// TwinCAT 3 PLC project Area2
// ProgramVersion: 3.1.4023.0
// libraries:
//   Tc2_DataExchange, * (Beckhoff Automation GmbH)
//   Tc2_EtherCAT, * (Beckhoff Automation GmbH)
//   Tc2_MC2, * (Beckhoff Automation GmbH)
//   Tc2_Standard, * (Beckhoff Automation GmbH)
//   Tc2_System, * (Beckhoff Automation GmbH)
//   Tc2_TcpIp, * (Beckhoff Automation GmbH)
//   Tc2_Utilities, * (Beckhoff Automation GmbH)
//   Tc3_BA_Common, * (Beckhoff Automation GmbH)
//   Tc3_Database, * (Beckhoff Automation GmbH)
//   Tc3_JsonXml, * (Beckhoff Automation GmbH)
//   Tc3_Module, * (Beckhoff Automation GmbH)
//   Tc3_PackML_V2, * (Beckhoff Automation GmbH)
// project tree:
//   COMs/Comms_ADS/ AdsData.TcDUT, AdsMessage.TcDUT, AdsMessageQueue.TcPOU, AdsSocket.TcPOU, AdsTcpUnitEx.TcPOU
//   COMs/Comms_TCP/ TcpServer1Vision.TcPOU (not stored), VisionFrame.TcDUT, VisionSuite.TcDUT
//   COMs/Comms_TCP/Types/ TcpData.TcDUT (not stored), TcpDataQueue.TcPOU (not stored)
//   COMs/Local Devices/ EcNetwork.TcPOU
//   COMs/ Watchdog.TcPOU
//   DUTs/Enums/ AreaEnum.TcDUT, E_PMLCustomUnitMode.TcDUT (not stored), SectionEnum.TcDUT, SectionTask.TcDUT, Cover.TcDUT (not stored), EventsEnum.TcTLEO, MaterialEnum.TcDUT, MaterialType.TcDUT (not stored), Surface.TcDUT (not stored)
//   DUTs/Enums/Materials/ Cardboard.TcDUT (not stored), Chipboard.TcDUT (not stored), CornerGuard.TcDUT (not stored), WoodBunk.TcDUT
//   DUTs/Hardware/ A21ToolStorage.TcDUT, FoldingMachine.TcDUT (not stored), PMLStackLight.TcPOU, ToolStorage.TcDUT
//   DUTs/Hardware/Big Machines/ StrapMachine.TcPOU, WrapMachine.TcPOU (not stored)
//   DUTs/Hardware/Conveyors/ Conveyor.TcPOU, ConveyorLSC.TcPOU (not stored), ConveyorMode.TcDUT (not stored), ConveyorSC.TcPOU, ConveyorSC_NC.TcPOU
//   DUTs/Hardware/Insertion Package/Drives/ AirPiston.TcPOU, ClearLinkMC.TcPOU (not stored), ServoNC.TcPOU, SimplePiston.TcPOU (not stored)
//   DUTs/Hardware/Insertion Package/ Homing.TcDUT (not stored), Insertion.TcPOU, SuctionPad.TcDUT
//   DUTs/Hardware/Insertion Package/Prototypes/ FBA_Drive.TcPOU (not stored), FBA_TrifectaDrive.TcPOU, I_ContinuousDrive.TcIO (not stored), I_Drive.TcIO, I_EncodedDrive.TcIO (not stored), I_PositionalDrive.TcIO
//   DUTs/Hardware/Material Holders/ MaterialHolder.TcPOU (not stored), MaterialSlot.TcDUT (not stored), SkidMagazine.TcPOU, StagingTable.TcPOU (not stored)
//   DUTs/Hardware/Robots/ I_Area2Robot.TcIO, KukaRobot.TcPOU, RobotA21.TcPOU, RobotA26.TcPOU, RobotA22.TcPOU
//   DUTs/Hardware/Robots/Tasks/ TaskA21.TcDUT (not stored), TaskA22.TcDUT (not stored), TaskA26.TcDUT
//   DUTs/Bundle/ Bundle.TcDUT, CardboardMaterial.TcDUT (not stored), Interval.TcDUT (not stored), Material.TcDUT (not stored), PositionMaterials.TcDUT
//   DUTs/Containers/ DynamicQueue.TcPOU (not stored), PtrQueue.TcPOU, IntQueue.TcPOU (not stored), Queue.TcPOU (not stored), StringQueue.TcPOU (not stored)
//   EventLogging/ EventLogger.TcIO (not stored), SqlDatabaseAccessor.TcPOU
//   / GlobalTextList.TcGTLO (not stored), PlcTask.TcTTO
//   GVLs/ COM.TcGVL, GVL.TcGVL, CONSTS.TcGVL
//   HARDWARE_DISTRUBUTION/ A24_A26.TcPOU, ConveyorSyncUnit.TcPOU, GenericSubarea.TcPOU, A21.TcPOU, A22.TcPOU, A23.TcPOU (not stored), A24.TcPOU, A25.TcPOU, A26.TcPOU (not stored)
//   POUs/Helper Functions/Document/ CreateJsonDocumentManual.TcPOU (not stored), CreateJsonDocumentAuto.TcPOU, FrameIsValid.TcPOU, VisionJsonParser.TcPOU (not stored)
//   POUs/Helper Functions/General/ BufferIsEmpty.TcPOU (not stored), BundleIsValid.TcPOU (not stored), InRange.TcPOU, PositionIsValid.TcPOU (not stored), TimestructToString.TcPOU (not stored), WithinTolerance.TcPOU
//   POUs/Helper Functions/Hardware Modules/ CheckEcNetwork.TcPOU, InsertionQuality.TcPOU, SetSuctions.TcPOU (not stored), SetSuctionsPtr.TcPOU (not stored), SetupHardware.TcPOU (not stored), SuctionQuality.TcPOU, SuctionQualityPtr.TcPOU (not stored)
//   POUs/Helper Functions/Material Functions/ GetPairMasterLength.TcPOU (not stored), GetMaterialLength.TcPOU, MatchesMaterialType.TcPOU
//   POUs/Helper Functions/Data Manipulation/ AddToStringArray.TcPOU, ArrayContains.TcPOU, DataIsEmpty.TcPOU (not stored), CleanStringsArray.TcPOU (not stored), IntegerBitAccess.TcPOU (not stored), IntegerToBoolArray.TcPOU (not stored), JoinStrings.TcPOU
//   POUs/ MAIN.TcPOU, TypeSizeCheck.TcPOU
//   Sections/A21a - Chipboard/AOIs/ AOI_LoadChipboard.TcPOU (not stored)
//   Sections/A21a - Chipboard/ ChipboardEx.TcPOU
//   Sections/A21b - Wood Bunk/AOIs/ AOI_LoadWoodBunk.TcPOU (not stored), AOI_StageWoodBunk.TcPOU, AOI_StagingTemplate.TcPOU (not stored)
//   Sections/A21b - Wood Bunk/ WoodBunkEx.TcPOU
//   Sections/A22 - Cardboard/AOIs/ AOI_LoadCornerCardboard.TcPOU (not stored), AOI_LoadCornerGuard.TcPOU (not stored), AOI_LoadFlatCardboard.TcPOU (not stored)
//   Sections/A22 - Cardboard/ CardboardEx.TcPOU
//   Sections/A26 - Spacer Recollection/ SpacerRecollectionUnit.TcPOU
//   Sections/Abstract/ SectionEx.TcPOU
// real-time tasks:
//   TASK PlcTask: cycle T#10ms, priority 20, ADS port 350
// motion (NC):
//   TASK NC-Task 1 SAF: cycle T#2ms, priority 4, ADS port 501
//   TASK NC-Task 1 SVB: cycle T#10ms, priority 8, ADS port 511
//   AXIS Axis 1 (id 1)
//     OtherSettings: AllowMotionCmdToSlave=true
//     encoder EncType=19
//       EncPara: MaxCount=#xffffffff
//     drive DrvType=16
//       DrvPara: MaxCount=#xffffffff, DriveControlDWord=#x00000100
//         Analog: TorqueSetpointScale=10, ScaleFactorActTorque=0.1
//         TimeComp: TaskDelayCycles=1
//     controller CtrType=1
//       CtrPara: PriorControlFactor=1
//         Observer: BandWidth=20
// I/O:
//   DEVICE Device 1 (EtherCAT) (disabled), AmsNetId 192.168.101.188.2.1
//     Term 1 (EK1200) [EK1200-5000 EtherCAT Power supply (2A E-Bus)]
//       Term 2 (EL2809) [EL2809 16Ch. Dig. Output 24V, 0.5A]
//       Term 3 (EL9011) [EL9011 End Terminal]
//   DEVICE Device 4 (EtherCAT) (disabled), AmsNetId 192.168.101.188.5.1
//     Drive 4 (CDHD) [CDHD EtherCAT Drive (CoE)]
// variable links:
//   NC-Task 1 SAF/Axes/Axis 1 <-> Device 4 (EtherCAT)/Drive 4 (CDHD)
//     Drive/Inputs/In/nDataIn1 <-> TxPDO 4/Following Error Actual Value
//     Drive/Inputs/In/nDataIn3[0] <-> TxPDO 1/Torque Actual Value
//     Drive/Inputs/In/nDcOutputTime <-> InfoData/DcOutputShift
//     Drive/Inputs/In/nState1 <-> TxPDO 1/StatusWord
//     Drive/Inputs/In/nState2 <-> TxPDO 1/StatusWord @bit 8
//     Drive/Inputs/In/nState4 @bit 1 <-> WcState/InputToggle
//     Drive/Inputs/In/nState4 <-> WcState/WcState
//     Drive/Inputs/In/nState5 <-> TxPDO 1/Modes of operation display
//     Drive/Outputs/Out/nCtrl1 <-> RxPDO 1/ControlWord
//     Drive/Outputs/Out/nCtrl2 <-> RxPDO 1/ControlWord @bit 8
//     Drive/Outputs/Out/nCtrl5 <-> RxPDO 1/Modes of operation
//     Drive/Outputs/Out/nDataOut1 <-> RxPDO 2/Target position
//     Drive/Outputs/Out/nDataOut2 <-> RxPDO 3/Target Velocity
//     Drive/Outputs/Out/nDataOut3[0] <-> RxPDO 4/Torque Offset
//     Drive/Outputs/Out/nDataOut4[0] <-> RxPDO 4/Target torque
//     Enc/Inputs/In/nDataIn1 <-> TxPDO 2/Position actual value
//     Enc/Inputs/In/nDcInputTime <-> InfoData/DcInputShift
//     Enc/Inputs/In/nState4 @bit 1 <-> WcState/InputToggle
//     Enc/Inputs/In/nState4 <-> WcState/WcState

CONFIGURATION Area2
    RESOURCE PLC ON TwinCAT3
        TASK PlcTask(INTERVAL := T#10ms, PRIORITY := 20);
        PROGRAM MAIN WITH PlcTask : MAIN;
    END_RESOURCE
END_CONFIGURATION

// ---- COMs/Comms_ADS/AdsData.TcDUT
{attribute 'enable_dynamic_creation'}
TYPE AdsData :
STRUCT
	description : EventsEnum; //purpose
	
	timestamp : TIMESTRUCT; //relevant timestamp (ex: arrival time)
	
	binaryData : ARRAY[0..100000] OF BYTE; //contents
END_STRUCT
END_TYPE

// ---- COMs/Comms_ADS/AdsMessage.TcDUT
{attribute 'enable_dynamic_creation'}
TYPE AdsMessage :
STRUCT
	recipient : STRING;
	contents : AdsData;
END_STRUCT
END_TYPE

// ---- COMs/Comms_TCP/VisionFrame.TcDUT
TYPE VisionFrame :
STRUCT
	MaterialID : STRING;
	CheckFor : STRING;
	CameraNumber : DINT;
	
	SuccessFlag : DINT;
	OrientAdjustX : LREAL;
	OrientAdjustY : LREAL;
	OrientAdjustZ : LREAL;
END_STRUCT
END_TYPE

// ---- COMs/Comms_TCP/VisionSuite.TcDUT
TYPE VisionSuite :
STRUCT
	json : STRING(1000);
	frame : VisionFrame;
	data : TcpData;
END_STRUCT
END_TYPE

// ---- DUTs/Enums/AreaEnum.TcDUT
{attribute 'qualified_only'}
{attribute 'to_string'}
TYPE AreaEnum :
(
	NULL_AREA,
	
	AREA_1,
	AREA_2,
	AREA_3,
	AREA_4,
	AREA_5,
	AREA_6,
	
	size
	
);
END_TYPE
(*
when generating AdsMessage types, use TO_STRING to convert these enums to a recipient string
*)

// ---- DUTs/Enums/Materials/WoodBunk.TcDUT
{attribute 'qualified_only'}
{attribute 'to_string'}
TYPE WoodBunk : //21
(
	WDW20 := 1, //special top (wide) 
	WDW22,

	WDT20, //top
	WDT22, 
	WDT28,

	WDB20, //bottom
	WDB22, 
	WDB28, 

	WDS08, //side
	WDS10, 
	WDS12, 
	WDS14, 
	WDS20, 
	WDS22, 
	WDS28, 
	
	size
	(*
	WDS08_WDS08, //side combined - X - 2 wood bunks joined by underscore
	WDS08_WDS10, 
	WDS12_WDS12, 
	WDS12_WDS14, 
	WDS20_WDS10, 
	WDS20_WDS12, 
	
	sizeAll
	*)
);
END_TYPE

// ---- DUTs/Enums/SectionEnum.TcDUT
{attribute 'qualified_only'}
{attribute 'to_string'}
TYPE SectionEnum :
(
	NULL_SECTION,
	
	PAPER,
	CARDBOARD_CORNERGUARD,
	CHIPBOARD,
	WOOD_BUNK,
	OUTPUT,
	
	SPACER_RECOLLECTOR,
	
	size
);
END_TYPE

// ---- DUTs/Hardware/A21ToolStorage.TcDUT
TYPE A21ToolStorage :
STRUCT
	pos1ChipboardEOAT AT %I* : BOOL;
	pos1WoodBunkEOAT AT %I* : BOOL;
	
	pos2ChipboardEOAT AT %I* : BOOL;
	pos2WoodBunkEOAT AT %I* : BOOL;
END_STRUCT
END_TYPE

// ---- DUTs/Hardware/Insertion Package/SuctionPad.TcDUT
TYPE SuctionPad :
STRUCT
	enable AT %Q* : BOOL;
	occupied AT %I* : BOOL;
END_STRUCT
END_TYPE

// ---- DUTs/Hardware/Robots/Tasks/TaskA26.TcDUT
{attribute 'qualified_only'}
{attribute 'to_string'}
//{attribute 'strict'}
TYPE TaskA26 :
(
	IDLE,
	PICK_SPACER,
	MEASURE,
	
	size
);
END_TYPE

// ---- DUTs/Hardware/ToolStorage.TcDUT
TYPE ToolStorage :
STRUCT
	eoatA_pos1 : BOOL;
	eoatB_pos1 : BOOL;
	
	eoatA_pos2 : BOOL;
	eoatB_pos2 : BOOL;	
END_STRUCT
END_TYPE

// ---- DUTs/Bundle/Bundle.TcDUT
{attribute 'enable_dynamic_creation'}
TYPE Bundle :
STRUCT
	id : STRING;
	weight : REAL;
	
	length : INT;
	width : INT;
	height : INT;
	
	pieces : INT;
	layers : INT;
	piecesPerLayer : INT;
	
	extrusionWeight : INT;
	extrusionHeight : INT;
	extrusionWidth : INT;
	
	//if a process is true, send it to the correct area and turn it false when complete
	reqProcesses : ARRAY[0..3] OF BOOL;
	
	manRE, autoRE : BOOL; //repacking - coming soon
	manSS, autoSS : BOOL; //packaging
	
	currStep : USINT; //for runtime use only
	
	paperFront : BOOL;
	paperBack : BOOL;
	cardboardFront : BOOL;
	cardboardBack : BOOL;
	
	paperTop : ARRAY[0..CONSTS.maxPairs] OF Interval;
	paperLeft : ARRAY[0..CONSTS.maxPairs] OF Interval;
	paperRight : ARRAY[0..CONSTS.maxPairs] OF Interval;
	paperBottom : ARRAY[0..CONSTS.maxPairs] OF Interval;
		
	cardboard : ARRAY[0..CONSTS.maxPairs] OF PositionMaterials;
	cardboardFolds : ARRAY[Surface.TOP_LEFT..Surface.BOTTOM_RIGHT] OF ARRAY[0..CONSTS.maxPairs] OF INT;
	
	topLeftFolds : ARRAY[0..CONSTS.maxPairs] OF INT;
	topRightFolds : ARRAY[0..CONSTS.maxPairs] OF INT;
	bottomLeftFolds : ARRAY[0..CONSTS.maxPairs] OF INT;
	bottomRightFolds : ARRAY[0..CONSTS.maxPairs] OF INT;
	
	cornerGuard : ARRAY[0..CONSTS.maxPairs] OF PositionMaterials;
	
	chipboard : ARRAY[0..CONSTS.maxPairs] OF PositionMaterials;
	woodBunk : ARRAY[0..CONSTS.maxPairs] OF PositionMaterials;
	
	cardboard_over_cornerGuard : BOOL;
	
	//for production log database
	bypass : BOOL;
	
	timeStart : TIMESTRUCT;
	timeDone : TIMESTRUCT;
END_STRUCT
END_TYPE

// ---- DUTs/Bundle/PositionMaterials.TcDUT
TYPE PositionMaterials : //REMOVE FOLDING INFORMATION FROM THIS STRUCTURE AND PLACE IN BUNDLE
STRUCT
	position : REAL; //:= GVL.nullPos; //default value is set to predefined constant if bundle needs less than 32 position material pairs
	
	top : STRING;
	right : STRING;
	left : STRING;
	//sides : STRING;
	bottom : STRING;
	
	topLeft : STRING;
	//topLeftFold : USINT;
	
	topRight : STRING;
	//topRightFold : USINT;
	
	bottomLeft : STRING;
	//bottomLeftFold : USINT;
	
	bottomRight : STRING;
	//bottomRightFold : USINT;

	wrapPoints : USINT;
	wrapRotations : USINT;
END_STRUCT
END_TYPE

// ---- DUTs/Enums/SectionTask.TcDUT
{attribute 'qualified_only'}
//{attribute 'strict'}
TYPE SectionTask :
(
	IDLE,
	ALIGNING,
	ACTIVE,
	DISCHARGE,
	COMPLETE,
	
	size
);
END_TYPE

// ---- DUTs/Enums/EventsEnum.TcTLEO
{attribute 'qualified_only'}
{attribute 'strict'}
{attribute 'to_string'}
TYPE EventsEnum :
(
	NO_EVENT,
	TEST_COMMS, 
	
	//standard operation
	BUNDLE_ETA,
	BUNDLE_IN,
	BUNDLE_OUT,
	BUNDLE_RECEIVED,
	BUNDLE_COMPLETE,
	
	//area complete
	AREA_1_COMPLETE,
	AREA_2_COMPLETE,
	AREA_3_COMPLETE,
	AREA_4_COMPLETE,
	AREA_5_COMPLETE,
	AREA_6_COMPLETE,
	
	//area specific operations
	SECTION_PAPER_COMPLETE,
	SECTION_CARDBOARD_CORNERGUARD_COMPLETE,
	SECTION_CHIPBOARD_COMPLETE,
	SECTION_WOODBUNK_COMPLETE,

	//standard errors
	BACKLOG,
	MACHINE_FAILURE,
	DELAY,
	BUNDLE_EARLY_RECEIVED,
	BUNDLE_LATE_RECEIVED,
	
	//area specific errors
	SECTION_PAPER_FAIL,
	SECTION_CARDBOARD_CORNERGUARD_FAIL,
	SECTION_CHIPBOARD_FAIL,
	SECTION_WOODBUNK_FAIL,
	
	//robots, motors, database, connections, etc
	
	size
);
END_TYPE

// ---- DUTs/Enums/MaterialEnum.TcDUT
{attribute 'qualified_only'}
{attribute 'strict'}
{attribute 'to_string'}
TYPE MaterialEnum :
(
	//CARDBOARD - 6 x 3
	CAR20S, CAR20M, CAR20L, CAR28S, CAR28M, CAR28L, //base (flat)
	CAR20SF, CAR20MF, CAR20LF, CAR28SF, CAR28MF, CAR28LF, //single folded (L shape) - F
	CAR20SD, CAR20MD, CAR20LD, CAR28SD, CAR28MD, CAR28LD, //double folded (C shape) - D
	
	//CHIPBOARD - 2
	CIP18, CIP54,
	
	//CORNER BOARD - 2
	COR48, COR96,
	
	//PAPER - 1
	PAP28,
	
	//WOOD BUNK - 21
	WDT20, WDT22, WDT28, //top
	WDB20, WDB22, WDB28, //bottom
	WDS08, WDS10, WDS12, WDS14, WDS20, WDS22, WDS28, //side
	WDS8X8, WDS8X10, WDS12X12, WDS12X14, WDS20X10, WDS20X12, //side combined - X
	WDW20, WDW22, //special top (wide)
	
	size //number of materials
);
END_TYPE

// ---- GVLs/COM.TcGVL
{attribute 'qualified_only'}
VAR_GLOBAL
	adsMajorNetwork : AdsTcpUnitEx;
END_VAR

// ---- GVLs/GVL.TcGVL
{attribute 'qualified_only'}
VAR_GLOBAL
	bundleOut : Bundle; //may or may not be used?
	
	iecCriticalSection : FB_IecCriticalSection; //if communication is separated into their own core/task
END_VAR
VAR_GLOBAL //changed from PROGRAMs to global instances of FUNCTION_BLOCKs to enable inheritance
	sa21 : A21;
	sa22 : A22;
	sa23 : A23;
	sa24 : A24;
	sa25 : A25;
	sa26 : A26;
END_VAR

// ---- GVLs/CONSTS.TcGVL
{attribute 'qualified_only'}
VAR_GLOBAL CONSTANT
	maxPairs : USINT := 16;
	initArraySize : USINT := 4;
	maxQueue : INT := 16;
	
	nullPos : REAL := -1;
	
	numMaterials : INT := 32;
	allMaterials : ARRAY[0..numMaterials] OF Material := [
		(code := '', width := 0, length := 0), //null material
		(code := 'PAP28', width := 28, length := -1),
		
		(code := 'CAR20S', width := 20, length := 30),
		(code := 'CAR20M', width := 20, length := 45),
		(code := 'CAR20L', width := 20, length := 60),
		(code := 'CAR28S', width := 28, length := 30),
		(code := 'CAR28M', width := 28, length := 45),
		(code := 'CAR28L', width := 28, length := 60),
		
		(code := 'COR48', width := 1.5, length := 48),
		(code := 'COR96', width := 1.5, length := 96),
		
		(code := 'CIP18', width := 20, length := 18),
		(code := 'CIP54', width := 20, length := 54),
		
		(code := 'WDT20', width := 20, length := 2.5),
		(code := 'WDT22', width := 22, length := 2.5),
		(code := 'WDT28', width := 28, length := 2.5),
		
		(code := 'WDB20', width := 20, length := 2.5),
		(code := 'WDB22', width := 22, length := 2.5),
		(code := 'WDB28', width := 28, length := 2.5),
		
		(code := 'WDS08', width := 8, length := 2.5),
		(code := 'WDS10', width := 10, length := 2.5),
		(code := 'WDS12', width := 12, length := 2.5),
		(code := 'WDS14', width := 14, length := 2.5),
		(code := 'WDS8x8', width := 16, length := 2.5),
		(code := 'WDS8x10', width := 18, length := 2.5),
		(code := 'WDS20', width := 20, length := 2.5),
		(code := 'WDS22', width := 22, length := 2.5),
		(code := 'WDS12x12', width := 24, length := 2.5),
		(code := 'WDS12x14', width := 26, length := 2.5),
		(code := 'WDS28', width := 28, length := 2.5),
		(code := 'WDS20x10', width := 30, length := 2.5),
		(code := 'WDS20x12', width := 32, length := 2.5),
		
		(code := 'WDW20', width := 20, length := 6),
		(code := 'WDW22', width := 22, length := 6)];
		
	precisionTolerance : REAL := 0.05 * 25.4;
END_VAR

// ---- DUTs/Hardware/Insertion Package/Prototypes/I_Drive.TcIO
INTERFACE I_Drive

{attribute 'monitoring':='call'}
PROPERTY Active : BOOL
GET
END_GET
END_PROPERTY

{attribute 'monitoring':='call'}
PROPERTY AtHome : BOOL
GET
END_GET
END_PROPERTY

{attribute 'monitoring':='call'}
PROPERTY Error : BOOL
GET
END_GET
END_PROPERTY

{attribute 'monitoring':='call'}
PROPERTY HomeSet : BOOL
GET
END_GET
END_PROPERTY

METHOD ABSTRACT homingSequence : BOOL
VAR_INPUT
END_VAR
END_METHOD

METHOD reset : BOOL
VAR_INPUT
END_VAR
END_METHOD

METHOD ABSTRACT stop : BOOL
VAR_INPUT
END_VAR
END_METHOD

METHOD toHome : BOOL
VAR_INPUT
END_VAR
END_METHOD

END_INTERFACE

// ---- DUTs/Hardware/Insertion Package/Prototypes/I_PositionalDrive.TcIO
INTERFACE I_PositionalDrive EXTENDS I_Drive

PROPERTY CurrentPosition : LREAL
GET
END_GET
SET
END_SET
END_PROPERTY

METHOD ABSTRACT moveAbsolute : BOOL
VAR_INPUT
	newTarget : LREAL; 
END_VAR
END_METHOD

METHOD ABSTRACT moveRelative : BOOL
VAR_INPUT
	distance : LREAL;
END_VAR
END_METHOD

PROPERTY TargetPosition : LREAL
GET
END_GET
SET
END_SET
END_PROPERTY

END_INTERFACE

// ---- DUTs/Hardware/Robots/I_Area2Robot.TcIO
INTERFACE I_Area2Robot
(*
currently all robots use 20-WORD arrays inputs and outputs so they extend from KukaRobot
if robot IOs are replaced with specific data types for each subarea, they should implement this interface instead
*)

//{attribute 'monitoring' := 'variable'}
{attribute 'monitoring' := 'call'}
PROPERTY Busy : BOOL
GET
END_GET
END_PROPERTY

METHOD clearCommand : BOOL
VAR_INPUT
END_VAR
END_METHOD

//{attribute 'monitoring' := 'variable'}
{attribute 'monitoring' := 'call'}
PROPERTY Done : BOOL
GET
END_GET
END_PROPERTY

{attribute 'monitoring' := 'call'}
PROPERTY Ready : BOOL
GET
END_GET
END_PROPERTY

METHOD release : BOOL
VAR_INPUT
	sectionReservation : SectionEnum;
END_VAR
END_METHOD

METHOD reserve : BOOL
VAR_INPUT
	reserveRequest : SectionEnum;
END_VAR
(*
this method exists because chipboard and wood bunk operations use the same robot
both sections need to check if the robot is open to commands before use
*)
END_METHOD

{attribute 'monitoring' := 'call'}
PROPERTY Reserved : BOOL
GET
END_GET
END_PROPERTY

METHOD reset : BOOL
END_METHOD

METHOD stop : BOOL
VAR_INPUT
END_VAR
END_METHOD

END_INTERFACE

// ---- POUs/MAIN.TcPOU
PROGRAM MAIN
VAR_OUTPUT //globally readable, but only modifiable by MAIN
	outputBufferPass, outputBufferFail : Bundle;
	numOutputBundles : USINT := 0;
	
	bundleIn : Bundle;
	bundleOut : Bundle;
	
	start : BOOL;
	
	ready : BOOL;
	busy : BOOL;
	done : BOOL;
	error : BOOL;
	backlog : BOOL;
	
	stop : BOOL;
	execute : BOOL;
	hold : BOOL;
	reset : BOOL;
	
	localTime : TIMESTRUCT;
	
	pmlMode : E_PMLCustomUnitMode;
	pmlState : E_PMLState;
	pmlModeString : STRING;
	pmlStateString : STRING;
END_VAR
VAR
	clearPassBuffer, clearFailBuffer AT %I* : BOOL;
	receiverStruct : AdsData;
	
	//ETA is not strictly required, area will process bundle even if it is not in ETA arrays
	expectedBundles : ARRAY[0..CONSTS.maxQueue] OF STRING; //bundles expected to arrive
	expectedArrivals : ARRAY[0..CONSTS.maxQueue] OF TIMESTRUCT; //bundles expected to arrive
	numEtaBundles : INT;
	
	//parallel arrays - bundle, bypass
	numBundles : INT;
	bundlesQueue : ARRAY[0..CONSTS.maxQueue] OF Bundle;
END_VAR
VAR //sections
	spacerRecollector : SpacerRecollectionUnit;
	//paperSection : PaperEx;
	cardboardSection : CardboardEx;
	chipboardSection : ChipboardEx;
	woodBunkSection : WoodBunkEx;
	//outputSection : AreaOutputEx;	
END_VAR
VAR
	ecDiagnostics_EK1200 : EcNetwork;
	
	fbLocalSystemTime : FB_LocalSystemTime;
	dbLogger : SqlDatabaseAccessor;
	
	pmlCommand : E_PMLCommand;
	pmlStateMachine : PML_StateMachine;
	
	pmlModeRequest : E_PMLCustomUnitMode := ePMLCustomUnitMode_Production;
	pmlModeManager : PML_UnitModeManager;
	
	processModes : (CONCURRENT, SINGLE, SERIAL);
	(*
	COCURRENT - cram as many bundles as can fit in the cell
	SINGLE - 1 bundle in the cell at a time, can be processed by many sections at the same time
	SERIAL - 1 bundle in the cell at a time, 1 section a time
		after completing a section, align bundle to action point of next section
	*)
END_VAR
VAR //these variables are only tracked for HMI
	sectionsBusy : ARRAY[0..SectionEnum.size] OF BOOL;
	sectionsIterator : ARRAY[0..SectionEnum.size] OF INT;
END_VAR
VAR
	cycleTime : DWORD;
	maxCycle : DWORD;
	masterProfiler : Profiler;
END_VAR

TypeSizeCheck();
masterProfiler(START:= TRUE, RESET:= , BUSY=> , DATA=> );

(*
Area 2 is ready when:
	no conveyors in A2.4 are occupied
	robot in A2.6 is not busy
if Area 2 is not ready, dispatch PLC must block operator from sending bundles here
*)

(*
busy := paperSection.busy OR cardboardCornerGuardSection.busy OR chipboardSection.busy OR woodBunkSection.busy OR outputSection.busy;
done := outputSection.done;
backlog := numBundlesQueue > 5;
*)

initSections();

blocks();

runPML();

runSubareas();

IF
	COM.adsMajorNetwork.fetchData(
		senderName := TO_STRING(AreaEnum.AREA_3), 
		data => receiverStruct)
THEN
	interpretTransmission(receiverStruct);
END_IF

IF ready AND BundleIsValid(bundleIn) THEN
	receive();
END_IF

IF clearPassBuffer OR clearFailBuffer THEN
	transfer();
	shiftBundles();
END_IF

dbLogger();

masterProfiler(START:= FALSE, RESET:= , BUSY=> , DATA=> );
cycleTime := masterProfiler.DATA.LastExecTime;
maxCycle := masterProfiler.DATA.MaxExecTime;

METHOD PRIVATE blocks : BOOL
fbLocalSystemTime(
	sNetID:= '', 
	bEnable:= TRUE, 
	dwCycle:= , 
	dwOpt:= , 
	tTimeout:= , 
	bValid=> , 
	systemTime=> localTime, 
	tzID=> );
	
ecDiagnostics_EK1200(
	enable:= TRUE, 
	netID:= , 
	slaves=> , 
	slaveStates=> , 
	deviceIndexesA21=> , 
	deviceIndexesA22=> , 
	deviceIndexesA23=> , 
	deviceIndexesA24=> , 
	deviceIndexesA25=> , 
	deviceIndexesA26=> , 
	numSlaves=> , 
	diagnosticsError=> ,
	errorInit=> , 
	errorPreop=> , 
	errorBootstrap=> , 
	errorSafeop=> , 
	operational=> );

ConveyorSyncUnit();
	
COM.adsMajorNetwork(
	setMode:= 1,
	bBusy=> , 
	error=> , 
	errorID=> );
	
TcpServer1Vision( //PLC-Vision comms
	ServerNetId:= , 
	ServerAdr:= , 
	ServerPort:= , 
	busy=> , 
	error=> , 
	errorId=> , 
	bytesReceived=> , 
	connected=> , 
	receiveStruct=> );
END_METHOD

METHOD fillBundlesQueue : BOOL
VAR
	i : INT;
END_VAR
IF NOT start THEN //for HMI testing only, remove for production
	FOR i:=0 TO CONSTS.maxQueue BY 1 DO
		bundlesQueue[i].id := TO_STRING(i);
	END_FOR
	
	start := TRUE;
END_IF
END_METHOD

METHOD PRIVATE initSections : BOOL
//paperSection.connectTo(ADR(cardboardCornerGuardSection));
//cardboardCornerGuardSection.connectTo(ADR(chipboardSection));
//chipboardSection.connectTo(ADR(woodBunkSection));
woodBunkSection.connectTo(0); //(ADR(outputSection));
//connecting to 0 means no next section

//paperSection.sectionID := SectionEnum.PAPER;
//cardboardCornerGuardSection.sectionID := SectionEnum.CARDBOARD_CORNERGUARD;
//chipboardSection.sectionID := SectionEnum.CHIPBOARD;
woodBunkSection.sectionID := SectionEnum.WOOD_BUNK;
//outputSection.sectionID := SectionEnum.OUTPUT;

(*
	paperSection.pNextSection := ADR(cardboardCornerGuardSection);
	cardboardCornerGuardSection.accessNextSection := ADR(chipboardSection);
	chipboardSection.accessNextSection := ADR(woodBunkSection);
	woodBunkSection.accessNextSection := ADR(outputSection);
	outputSection.accessNextSection := 0;
*)

initSections := TRUE;
END_METHOD

METHOD PRIVATE interpretTransmission : BOOL
VAR_INPUT
	data : REFERENCE TO AdsData;
END_VAR
VAR
	i : INT;
END_VAR
CASE data.description OF
	EventsEnum.BUNDLE_IN:
		MEMCPY(ADR(bundleIn), ADR(data.binaryData), SIZEOF(bundleIn));
			
	EventsEnum.BUNDLE_ETA:
		MEMCPY(ADR(expectedBundles[numEtaBundles]), ADR(data.binaryData), SIZEOF(expectedBundles[numEtaBundles]));
		expectedArrivals[numEtaBundles] := data.timestamp;
		
END_CASE
END_METHOD

METHOD maintenance : BOOL
VAR_INPUT
END_VAR
END_METHOD

METHOD PRIVATE process : BOOL
(*
full parallel processsing
all sections may operate concurrently on any bundle
*)
(*
paperSection(
	enable:= run[SectionEnum.PAPER], 
	bundlesQueue:= bundlesQueue, 
	bundlesBypass:= bundlesBypass,
	bundleOut=> , 
	bypass=> , 
	ready=> , 
	busy=> sectionsBusy[SectionEnum.PAPER], 
	done=> , 
	error=> , 
	backlog=> ,
	iBundle=> sectionsIterator[SectionEnum.PAPER],
	iPair=> );
	
cardboardCornerGuardSection(
	enable:= run[SectionEnum.CARDBOARD_CORNERGUARD],
	bundlesQueue:= bundlesQueue, 
	bundlesBypass:= bundlesBypass,
	bundleOut=> ,
	bypass=> , 
	ready=> , 
	busy=> sectionsBusy[SectionEnum.CARDBOARD_CORNERGUARD], 
	done=> , 
	error=> , 
	backlog=> ,
	iBundle=> sectionsIterator[SectionEnum.CARDBOARD_CORNERGUARD],
	iPair=> );

chipboardSection(
	enable:= run[SectionEnum.CHIPBOARD],
	bundlesQueue:= bundlesQueue, 
	bundlesBypass:= bundlesBypass, 
	bundleOut=> ,
	bypass=> , 
	ready=> , 
	busy=> sectionsBusy[SectionEnum.CHIPBOARD], 
	done=> , 
	error=> , 
	backlog=> ,
	iBundle=> sectionsIterator[SectionEnum.CHIPBOARD],
	iPair=> );
*)

(*
woodBunkSection(
	enable:= run[SectionEnum.WOOD_BUNK],
	bundlesQueue:= bundlesQueue, 
	bundlesBypass:= bundlesBypass, 
	bundleOut=> ,
	bypass=> , 
	ready=> , 
	busy=> sectionsBusy[SectionEnum.WOOD_BUNK], 
	done=> , 
	error=> , 
	backlog=> ,
	iBundle=> sectionsIterator[SectionEnum.WOOD_BUNK],
	iPair=> );
*)
(*
outputSection(
	enable:= run[SectionEnum.OUTPUT],
	bundlesQueue:= bundlesQueue, 
	bundlesBypass:= bundlesBypass,
	outputBuffer:= outputBuffer,
	bundleOut=> , 
	bypass=> , 
	ready=> , 
	busy=> sectionsBusy[SectionEnum.OUTPUT],
	done=> , 
	error=> , 
	backlog=> ,
	iBundle=> sectionsIterator[SectionEnum.OUTPUT],
	iPair=> );
*)
END_METHOD

METHOD PRIVATE ps_AbortCondition : BOOL
VAR_INPUT
END_VAR
END_METHOD

METHOD PRIVATE ps_Aborted : BOOL
VAR_INPUT
END_VAR
END_METHOD

METHOD PRIVATE ps_Aborting : BOOL
VAR_INPUT
END_VAR
END_METHOD

METHOD PRIVATE ps_Clearing : BOOL
VAR_INPUT
END_VAR
END_METHOD

METHOD PRIVATE ps_Complete : BOOL
VAR_INPUT
END_VAR
END_METHOD

METHOD PRIVATE ps_Completing : BOOL
VAR_INPUT
END_VAR
END_METHOD

METHOD PRIVATE ps_Execute : BOOL
VAR_INPUT
END_VAR
VAR_OUTPUT
	error : BOOL;
END_VAR
CASE pmlMode OF
	0: //invalid mode
	ePMLCustomUnitMode_Production:		ps_Execute := process();
	ePMLCustomUnitMode_Maintenance:		maintenance();
	ePMLCustomUnitMode_Manual:			//
	ePMLCustomUnitMode_SemiAuto:		ps_Execute := process(); //manually step bundle into area - sections may be auto while area is semi-auto
END_CASE
END_METHOD

METHOD PRIVATE ps_Held : BOOL
VAR_INPUT
END_VAR
END_METHOD

METHOD PRIVATE ps_HoldCondition : BOOL
VAR_INPUT
END_VAR
END_METHOD

METHOD PRIVATE ps_Holding : BOOL
VAR_INPUT
END_VAR
END_METHOD

METHOD PRIVATE ps_Idle : BOOL
VAR_INPUT
END_VAR
(*
IF BundleIsValid(currentBundle) THEN
	ps_Idle := TRUE;
	done := FALSE;
END_IF
*)

ps_Idle := TRUE; (*start section input*)
END_METHOD

METHOD PRIVATE ps_Resetting : BOOL
VAR_INPUT
END_VAR
END_METHOD

METHOD PRIVATE ps_Starting : BOOL
VAR_INPUT
END_VAR
END_METHOD

METHOD PRIVATE ps_StopCondition : BOOL
VAR_INPUT
END_VAR
END_METHOD

METHOD PRIVATE ps_Stopped : BOOL
VAR_INPUT
END_VAR
END_METHOD

METHOD PRIVATE ps_Stopping : BOOL
VAR_INPUT
END_VAR
END_METHOD

METHOD PRIVATE ps_SuspendCondition : BOOL
VAR_INPUT
END_VAR
END_METHOD

METHOD PRIVATE ps_Suspended : BOOL
VAR_INPUT
END_VAR
END_METHOD

METHOD PRIVATE ps_Suspending : BOOL
VAR_INPUT
END_VAR
END_METHOD

METHOD PRIVATE ps_Unholding : BOOL
VAR_INPUT
END_VAR
END_METHOD

METHOD PRIVATE ps_Unsuspending : BOOL
VAR_INPUT
END_VAR
END_METHOD

{attribute 'TcRpcEnable'}
METHOD PRIVATE receive : BOOL
VAR
	i : INT;
	etaIndex : INT := -1;
END_VAR
FOR i:=0 TO CONSTS.maxQueue BY 1 DO //find the bundle in the ETA queue
	IF expectedBundles[i] = bundleIn.id THEN
		etaIndex := i;
		EXIT;
	END_IF
END_FOR

IF etaIndex > -1 THEN //if the bundle is found in the ETA queue, shift everything down
	MEMMOVE(
		ADR(expectedBundles[etaIndex]), 
		ADR(expectedBundles[MAX(etaIndex + 1, CONSTS.maxQueue)]), 
		SIZEOF(STRING) * TO_UINT(CONSTS.maxQueue - etaIndex));
		
	MEMMOVE(
		ADR(expectedArrivals[etaIndex]), 
		ADR(expectedArrivals[MAX(etaIndex + 1, CONSTS.maxQueue)]), 
		SIZEOF(TIMESTRUCT) * TO_UINT(CONSTS.maxQueue - etaIndex) );
		
	MEMSET(ADR(expectedBundles[CONSTS.maxQueue]), 0, SIZEOF(expectedBundles[0]));
	MEMSET(ADR(expectedArrivals[CONSTS.maxQueue]), 0, SIZEOF(expectedArrivals[0]));	
		
	numEtaBundles := numEtaBundles - 1;
END_IF

FOR i:=0 TO CONSTS.maxQueue BY 1 DO
	IF NOT BundleIsValid(bundlesQueue[i]) THEN
		bundlesQueue[i] := bundleIn;
		
		receive := TRUE;
		RETURN;
	END_IF
END_FOR

IF NOT receive THEN
	error := TRUE;
END_IF
END_METHOD

METHOD PRIVATE runPML : BOOL
(*
PackML
	state machine for packaging applications - see Tc3_PackML_V2 library on InfoSys
	
	final states - wait for an input or condition and command to new state
	intermediate states - complete a task and call pmlStateMachine.M_StateComplete() to advance to next state
	
the following states currently use the same logic (albeit in different methods), implementation may change later
	ps_Stopping() and ps_Aborting()
	ps_Resetting() and ps_Clearing()
	
STOP - controlled stop **with intent to shutdown or vacate for extended time** induced by operator/HMI - otherwise use HOLD
ABORT - emergency stop due to machine errors


HOLD - minor local issues
SUSPEND - external issues

EXECUTE - major control logic
	different modes may require different tasks
	create methods as required for different modes, then call the correct method in ps_Completing()
	can be commanded to STOP, ABORT, HOLD, or SUSPEND at any point
COMPLETING - process complete, move product out of system and finish transition to COMPLETED

the implementation below can be copied to all POUs that use a PackML state machine
the individual ps_< > methods need to be implemented for the specific application
*)
IF ps_AbortCondition() THEN //abort condition
	pmlCommand := ePMLCommand_Abort;
ELSIF ps_StopCondition() THEN //stop condition
	pmlCommand := ePMLCommand_Stop;
END_IF

CASE pmlState OF
	0 (*ePMLState_Undefined*): //default state on startup
		pmlCommand := ePMLCommand_Stop;
		
	ePMLState_Stopping:
		IF ps_Stopping() THEN
			pmlStateMachine.M_StateComplete();
		END_IF
		
	ePMLState_Stopped:
		IF ps_Stopped() THEN
			pmlCommand := ePMLCommand_Reset;
		END_IF
	
    ePMLState_Resetting:
		IF ps_Resetting() THEN
			pmlStateMachine.M_StateComplete();
		END_IF
		
	ePMLState_Idle:
		IF ps_Idle() THEN
			pmlCommand := ePMLCommand_Start;
		END_IF		
	
	ePMLState_Starting:
		IF ps_Starting() THEN
			pmlStateMachine.M_StateComplete();
		END_IF
	
	ePMLState_Execute: //check the conditions in order of their priority, currently HOLD has the highest priority
		IF ps_HoldCondition() THEN
			pmlCommand := ePMLCommand_Hold;
			
		ELSIF ps_SuspendCondition() THEN
			pmlCommand := ePMLCommand_Suspend;			
		
		ELSIF ps_Execute(error => error) THEN //ps_Execute.error => THIS^.error
			pmlStateMachine.M_StateComplete();
			pmlCommand := ePMLCommand_Complete;
		END_IF
		
	ePMLState_Completing:
		IF ps_Completing() THEN
			pmlStateMachine.M_StateComplete();
		END_IF
	
	ePMLState_Complete:
		IF ps_Complete() THEN
			pmlCommand := ePMLCommand_Reset;
		END_IF
	
	ePMLState_Holding:
		IF ps_Holding() THEN
			pmlStateMachine.M_StateComplete();
		END_IF
	
	ePMLState_Held:
		IF NOT hold THEN
			pmlCommand := ePMLCommand_Unhold;
		END_IF
	
	ePMLState_Unholding:
		IF ps_Unholding() THEN
			pmlStateMachine.M_StateComplete(); //release all pause commands and IO
		END_IF
		
	ePMLState_Suspending: //based on next section conditions
		IF ps_Suspending() THEN
			pmlStateMachine.M_StateComplete();
		END_IF
		
	ePMLState_Suspended: //based on next section conditions
		IF ps_Suspended() THEN
			pmlCommand := ePMLCommand_Unsuspend;
		END_IF
	
	ePMLState_Unsuspending: //based on next section conditions
		IF ps_Unsuspending() THEN
			pmlStateMachine.M_StateComplete();
		END_IF
	
	ePMLState_Aborting:
		IF ps_Aborting() THEN
			pmlStateMachine.M_StateComplete();
		END_IF
	
	ePMLState_Aborted:
		IF ps_Aborted() THEN
			pmlCommand := ePMLCommand_Clear;
		END_IF
	
	ePMLState_Clearing:
		IF ps_Clearing() THEN
			pmlStateMachine.M_StateComplete();
		END_IF
	
END_CASE
END_METHOD

METHOD PRIVATE runSubareas : BOOL
(*
the new program structure specifies the following:
	declare the section modules in MAIN,
	declare the hardware modules in the approrpiate subarea module
		see folder HARDWARE_DISTRIBUTION for all 6 subareas
	pass the section modules to one of the 6 subarea hardware distrubutors to be called with their required hardware
	
conveyors are declared in ConveyorSyncUnit as VAR_OUTPUTs to be made visible without tying them to any specific subarea

this structure should drastically reduce the visibility of hardware modules and eliminate the need for large GVLs
*)
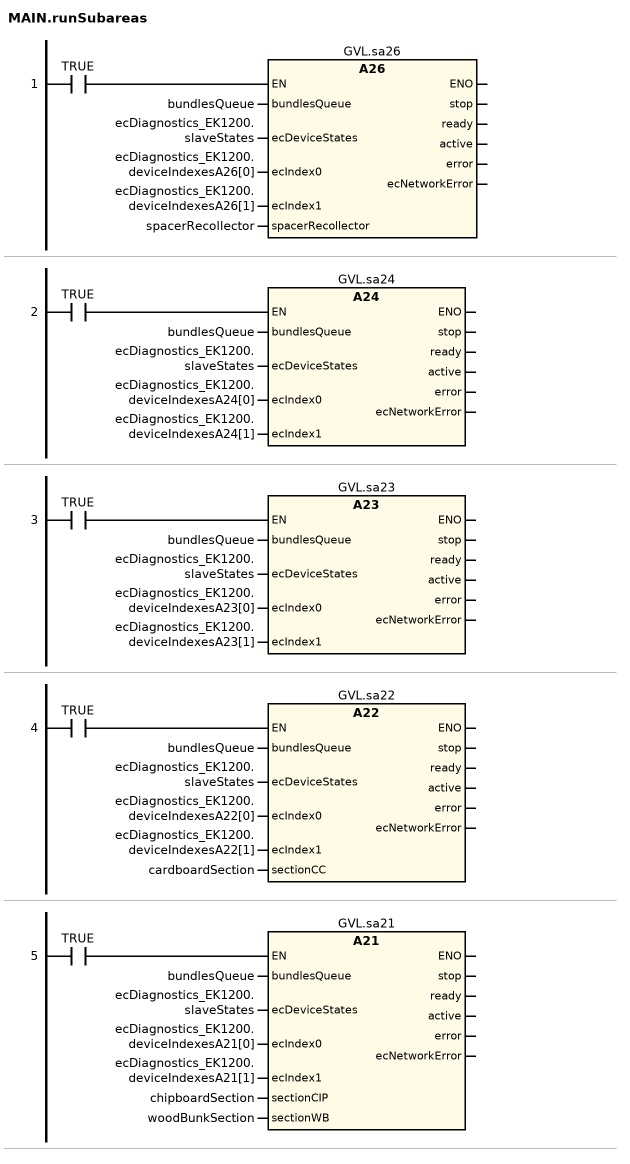
// NETWORK 1
GVL.sa26(
    bundlesQueue := bundlesQueue,
    ecDeviceStates := ecDiagnostics_EK1200.slaveStates,
    ecIndex0 := ecDiagnostics_EK1200.deviceIndexesA26[0],
    ecIndex1 := ecDiagnostics_EK1200.deviceIndexesA26[1],
    spacerRecollector := spacerRecollector); // A26

// NETWORK 2
GVL.sa24(
    bundlesQueue := bundlesQueue,
    ecDeviceStates := ecDiagnostics_EK1200.slaveStates,
    ecIndex0 := ecDiagnostics_EK1200.deviceIndexesA24[0],
    ecIndex1 := ecDiagnostics_EK1200.deviceIndexesA24[1]); // A24

// NETWORK 3
GVL.sa23(
    bundlesQueue := bundlesQueue,
    ecDeviceStates := ecDiagnostics_EK1200.slaveStates,
    ecIndex0 := ecDiagnostics_EK1200.deviceIndexesA23[0],
    ecIndex1 := ecDiagnostics_EK1200.deviceIndexesA23[1]); // A23

// NETWORK 4
GVL.sa22(
    bundlesQueue := bundlesQueue,
    ecDeviceStates := ecDiagnostics_EK1200.slaveStates,
    ecIndex0 := ecDiagnostics_EK1200.deviceIndexesA22[0],
    ecIndex1 := ecDiagnostics_EK1200.deviceIndexesA22[1],
    sectionCC := cardboardSection); // A22

// NETWORK 5
GVL.sa21(
    bundlesQueue := bundlesQueue,
    ecDeviceStates := ecDiagnostics_EK1200.slaveStates,
    ecIndex0 := ecDiagnostics_EK1200.deviceIndexesA21[0],
    ecIndex1 := ecDiagnostics_EK1200.deviceIndexesA21[1],
    sectionCIP := chipboardSection,
    sectionWB := woodBunkSection); // A21
END_METHOD

METHOD shiftBundles : BOOL
VAR_INPUT
END_VAR
//shift down bundles queue
MEMMOVE(ADR(bundlesQueue[0]), ADR(bundlesQueue[1]), SIZEOF(Bundle) * TO_UINT(CONSTS.maxQueue));

//decrement each section's iterator to realign with their correct bundle
//paperSection.shiftIterator();
//cardboardCornerGuardSection.shiftIterator();
chipboardSection.shiftIterator();
woodBunkSection.shiftIterator();
//outputSection.shiftIterator();
END_METHOD

METHOD PRIVATE transfer : BOOL
VAR
	i : INT;
END_VAR
//send TCP/ADS transmission back to Dispatch once bundle is removed from the plant

IF clearPassBuffer THEN
	dbLogger.queueEvent(event:= EventsEnum.BUNDLE_OUT); //modify to include bundle ID
	//outputBufferPass := GVL.nullBundle;
	MEMSET(ADR(outputBufferPass), 0, SIZEOF(outputBufferPass));
END_IF

IF clearFailBuffer THEN
	dbLogger.queueEvent(event:= EventsEnum.BUNDLE_OUT); //modify to include bundle ID
	//outputBufferFail := GVL.nullBundle;
	MEMSET(ADR(outputBufferFail), 0, SIZEOF(outputBufferFail));
END_IF
END_METHOD

END_PROGRAM

// ---- Sections/A26 - Spacer Recollection/SpacerRecollectionUnit.TcPOU
FUNCTION_BLOCK SpacerRecollectionUnit //EXTENDS SectionEx
VAR_IN_OUT
	robot : RobotA26;
	robotSlider : ServoNC;
	(*
	A24_LRC_C01 : Conveyor;
	A24_LRC_C03 : Conveyor;
	A24_LRC_C05 : Conveyor;
	A24_LRC_C07 : Conveyor;
	A24_LRC_C09 : Conveyor;
	A24_LRC_C11 : Conveyor;
	A24_LRC_C13 : Conveyor;
	
	A24_LRC_C02 : ConveyorSC;
	A24_LRC_C04 : ConveyorSC;
	A24_LRC_C06 : ConveyorSC;
	A24_LRC_C08 : ConveyorSC;
	A24_LRC_C10 : ConveyorSC;
	A24_LRC_C12 : ConveyorSC;
	*)
END_VAR
VAR_INPUT
	conveyorOccupied_A24_LRC_C01 : BOOL; //odd number conveyors move the conveyor down the cell
	conveyorOccupied_A24_LRC_C03 : BOOL;
	conveyorOccupied_A24_LRC_C05 : BOOL;
	conveyorOccupied_A24_LRC_C07 : BOOL;
	conveyorOccupied_A24_LRC_C09 : BOOL;
	conveyorOccupied_A24_LRC_C11 : BOOL;
	conveyorOccupied_A24_LRC_C13 : BOOL;
	
	spacerPresent_A24_LRC_C02 : BOOL;
	spacerPresent_A24_LRC_C04 : BOOL;
	spacerPresent_A24_LRC_C06 : BOOL;
	spacerPresent_A24_LRC_C08 : BOOL;
	spacerPresent_A24_LRC_C10 : BOOL;
	spacerPresent_A24_LRC_C12 : BOOL;
END_VAR
VAR_OUTPUT
	ready : BOOL;
	busy : BOOL;
	done : BOOL;
	error : BOOL;
	
	failCounter : INT;
END_VAR
VAR
	status : SectionTask;
	step : (IDLE, SLIDE, PICK_SPACER);
	iConveyorLine : INT;
END_VAR
VAR //slider positions
	pickPos1, pickPos2 : LREAL;
END_VAR
VAR_STAT CONSTANT
	COMPLETE : INT := 1050;
END_VAR

ready := step = 0;
busy := step > 0;
done := done;
error := error;

CASE status OF
	SectionTask.IDLE: //do nothing
	
	SectionTask.ALIGN: //receive incoming bundle
	
	SectionTask.ACTIVE: //measure new bundle
		
	SectionTask.DISCHARGE: //send bundle down cell, then clear spacers
		IF 
			conveyorOccupied_A24_LRC_C01 OR
			conveyorOccupied_A24_LRC_C03 OR
			conveyorOccupied_A24_LRC_C05 OR
			conveyorOccupied_A24_LRC_C07 OR
			conveyorOccupied_A24_LRC_C09 OR
			conveyorOccupied_A24_LRC_C11 OR
			conveyorOccupied_A24_LRC_C13
		THEN
			
			robot.clearCommand();
			
		ELSIF process() THEN //remove spacers from transfer conveyors in ascending order
			status := SectionTask.COMPLETE;
			
		END_IF
		
	SectionTask.COMPLETE: //reset, ready to receive next bundle
		done := TRUE;
	
END_CASE

METHOD process : BOOL
VAR
	spacersPresent : ARRAY[1..6] OF BOOL := [
		spacerPresent_A24_LRC_C02,
		spacerPresent_A24_LRC_C04,
		spacerPresent_A24_LRC_C06,
		spacerPresent_A24_LRC_C08,
		spacerPresent_A24_LRC_C10,
		spacerPresent_A24_LRC_C12];
END_VAR
VAR CONSTANT
	suctionDistance : INT := 10;
END_VAR
{warning disable C0371}

iConveyorLine := MAX(1, iConveyorLine); //value is always at least 1

CASE step OF
	IDLE:
		IF DataIsEmpty(arr := ADR(spacersPresent), arrSize := SIZEOF(spacersPresent)) THEN
			robotSlider.toHome();
			
			iConveyorLine := 0;
			failCounter := 0;
			process := TRUE;
		
		ELSIF NOT spacersPresent[iConveyorLine] THEN
			iConveyorLine := iConveyorLine + 1;
			
		ELSIF robot.Ready THEN
			step := SLIDE;
			
		END_IF
		
	SLIDE:
		CASE iConveyorLine OF
			1,2,3:		robotSlider.moveAbsolute(newTarget := pickPos1);
			4,5,6:		robotSlider.moveAbsolute(newTarget := pickPos2);
		END_CASE
		
		//replace this condition with WithinTolerance() if the slider spends too long adjusting its position
		IF robotSlider.CurrentPosition = robotSlider.TargetPosition THEN
			step := PICK_SPACER;
		END_IF
		
	PICK_SPACER:		
		IF robot.eoatDistance > suctionDistance THEN
			robot.HoldMaterial := 'SPACER';
		ELSE
			robot.HoldMaterial := '';
		END_IF
	
		IF robot.Done THEN
			step := COMPLETE;
		ELSE
			robot.setGroup(group := 1, value := TaskA26.PICK_SPACER);
			robot.setGroup(group := 2, value := iConveyorLine);
		END_IF
		
	COMPLETE:
		robot.HoldMaterial := '';
		
		IF spacersPresent[iConveyorLine] THEN
			failCounter := failCounter + 1;
		END_IF
		
		robot.clearCommand();
		step := 0;
	
END_CASE
END_METHOD

END_FUNCTION_BLOCK

// ---- DUTs/Hardware/Robots/RobotA26.TcPOU
FUNCTION_BLOCK RobotA26 EXTENDS KukaRobot
VAR_INPUT
	conveyorSafety : BOOL;
END_VAR
VAR_OUTPUT //from outputs array
	{warning disable C0195}
	taskID : TaskA26;
	param1 : INT; //position number (1..6)
	param2 : INT;
	
	strapSafetyOut : BOOL;
END_VAR
VAR_OUTPUT //from inputs array
	tool : SectionEnum := SectionEnum.SPACER_RECOLLECTOR;
	suspendedMaterial : STRING;
	
	completedTask : TaskA26;
	eoatDistance : INT;
	
	conveyorSafetyIn : BOOL;
END_VAR
VAR
	reservationEnum : SectionEnum;
	hmiTask : STRING;
	hmiTool : STRING;
END_VAR
(*
extends KukaRobot
	assigns descriptive labels to each IO group from the array
	additional section-specific methods to get/set IO groups
*)

(*
parameters - aliases to IO elements
command - full IO array
*)
{warning disable C0195}
SUPER^();

outputs[1] := taskID;
outputs[2] := param1;
outputs[3] := param2;

outputs[8].15 := conveyorSafety;

refreshParameters();

reservationEnum := reservation;
IF reservationEnum = SectionEnum.NULL_SECTION THEN
	hmiReservation := 'N/A';
ELSE
	hmiReservation := TO_STRING(reservationEnum);
END_IF

hmiTask := TO_STRING(taskID);
hmiTool := TO_STRING(tool);

{attribute 'monitoring' := 'call'}
PROPERTY Busy : BOOL
GET
VAR
	//emptyOutput : ARRAY[1..50] OF INT;
END_VAR
//Busy stays TRUE until outputs are cleared AND completed task has elapsed
//Ready is always inverse of Busy
refreshParameters();

Busy := taskID <> 0 OR completedTask <> 0;
END_GET
END_PROPERTY

METHOD clearCommand : BOOL
VAR_INPUT
END_VAR
SUPER^.clearCommand();

refreshParameters();
END_METHOD

{attribute 'monitoring' := 'call'}
PROPERTY Done : BOOL
GET
refreshParameters();

Done :=
	completedTask = taskID AND
	taskID <> 0 AND
	completedTask <> 0;
END_GET
END_PROPERTY

{attribute 'monitoring' := 'call'}
PROPERTY HoldMaterial : STRING
GET
HoldMaterial := suspendedMaterial;
END_GET
SET
suspendedMaterial := HoldMaterial;
END_SET
END_PROPERTY

{attribute 'monitoring' := 'call'}
PROPERTY Ready : BOOL
GET
refreshParameters();

Ready := taskID = 0 AND completedTask = 0 AND NOT error;
END_GET
END_PROPERTY

METHOD PRIVATE refreshParameters : BOOL
VAR_INPUT
END_VAR
{warning disable C0196}
taskID := outputs[1];
param1 := outputs[2];
param2 := outputs[3];

conveyorSafetyIn := inputs[4].15;
END_METHOD

METHOD setGroup : BOOL
VAR_INPUT
	group : INT;
	value : INT;
END_VAR
SUPER^.setGroup(group := group, value := value);

refreshParameters();
END_METHOD

METHOD setParameters : BOOL
VAR_INPUT
	newTaskID : INT;
	newParam1 : INT;
	newParam2 : INT;
	newXmm : INT;
	newYmm : INT;
	newZmm : INT;
	newAngle : INT;
	newStagingOccupancy : INT;
	newInsertionSuctionStatus : INT;
	newMagazineStatus : INT; //unused
	newInspectionValue : INT;
END_VAR
VAR_INPUT
	strapSafety : BOOL;
END_VAR
setGroup(group := 1, value := newTaskID);
setGroup(group := 2, value := newParam1);
setGroup(group := 3, value := newParam2);

refreshParameters();
END_METHOD

END_FUNCTION_BLOCK

// ---- DUTs/Hardware/Robots/KukaRobot.TcPOU
FUNCTION_BLOCK KukaRobot
VAR_INPUT
	bEnable : BOOL; //this enables the robot
	abort : BOOL; //this disables the robot
	//bEnable must be TRUE and abort must be FALSE for the robot to function
END_VAR
VAR_OUTPUT
	(*
	forceStop AT %Q* : BOOL;
	resetSignal AT %Q* : BOOL;
	*)
	
	reservation : INT := 0;
	
	error : BOOL;
	errId : DINT;
	
	outputs AT %Q* : ARRAY[1..20] OF WORD;
	inputs AT %I* : ARRAY[1..20] OF WORD;
END_VAR
VAR
	heartbeat : Watchdog;
	
	toggleBit AT %I* : BOOL; //check connection from PLC to bridge
	disconnected AT %I* : BOOL; //check connection from bridge to robot
	
	hmiReservation : STRING;
END_VAR
(*
generic KUKA robot with 20 WORD outputs and 20 WORD inputs, connected to Beckhoff IPC via EL6692 or EL6695 EtherCAT bridge
includes minimal diagnostics to detect if robot is offline
robots should always be reserved before sending a task
*)

heartbeat(
	enable:= NOT disconnected,
	toggleBit:= toggleBit,
	timeoutWidth:= T#200MS,
	timeout=> );

error := //add any addition conditions with OR
	disconnected OR
	heartbeat.timeout;
	
IF (*NOT bEnable OR*) abort THEN //bEnable is not used for now, but abort is
	stop();
END_IF

//{attribute 'monitoring' := 'variable'}
{attribute 'monitoring' := 'call'}
PROPERTY Busy : BOOL
GET
END_GET
END_PROPERTY

METHOD clearCommand : BOOL
VAR_INPUT
END_VAR
MEMSET(ADR(outputs), 0, SIZEOF(outputs));
END_METHOD

//{attribute 'monitoring' := 'variable'}
{attribute 'monitoring' := 'call'}
PROPERTY Done : BOOL
GET
END_GET
END_PROPERTY

{attribute 'monitoring' := 'call'}
PROPERTY Ready : BOOL
GET
END_GET
END_PROPERTY

METHOD release : BOOL
VAR_INPUT
	sectionReservation : SectionEnum;
END_VAR
IF reservation = sectionReservation THEN
	reservation := SectionEnum.NULL_SECTION;
	release := TRUE;
END_IF
END_METHOD

METHOD reserve : BOOL
VAR_INPUT
	reserveRequest : SectionEnum;
END_VAR
(*
this method exists because chipboard and wood bunk operations use the same robot
both sections need to check if the robot is open to commands before use
*)
IF Reserved AND reservation = reserveRequest THEN
	reserve := TRUE;

ELSIF NOT Reserved THEN
	reservation := reserveRequest;
	reserve := TRUE;

END_IF
END_METHOD

{attribute 'monitoring' := 'call'}
PROPERTY Reserved : BOOL
GET
Reserved := reservation <> SectionEnum.NULL_SECTION;
END_GET
END_PROPERTY

METHOD reset : BOOL
//resetSignal := TRUE;
//done := FALSE;

MEMSET(ADR(outputs), 0, SIZEOF(outputs));
(*
IF ready AND completedTask = 0 THEN
	resetSignal := FALSE;
	reset := TRUE;
END_IF
*)
END_METHOD

METHOD resume : BOOL
VAR_INPUT
END_VAR
//forceStop := FALSE;

resume := NOT error AND errId = 0;
END_METHOD

METHOD setGroup : BOOL
VAR_INPUT
	group : INT;
	value : INT;
END_VAR
{warning disable C0195}
outputs[group] := value;
END_METHOD

METHOD stop : BOOL
VAR_INPUT
END_VAR
//forceStop := TRUE;
clearCommand();

stop := TRUE;
END_METHOD

END_FUNCTION_BLOCK

// ---- COMs/Watchdog.TcPOU
FUNCTION_BLOCK Watchdog
VAR_INPUT
	enable : BOOL := TRUE; //watchdog can be disabled if needed
	
	toggleBit : BOOL;
	timeoutWidth : TIME := DEFAULT_ADS_TIMEOUT;
END_VAR
VAR_OUTPUT
	timeout : BOOL;
	prevMsgTimestamp : TIMESTRUCT;
END_VAR
VAR	
	timer : TON;
	memoryBit : BOOL;
END_VAR

timer(
	IN:= enable AND (memoryBit = toggleBit), 
	PT:= timeoutWidth, 
	Q=> timeout, 
	ET=> );
	
IF enable AND memoryBit <> toggleBit THEN
	prevMsgTimestamp := MAIN.localTime;
END_IF

memoryBit := toggleBit;

END_FUNCTION_BLOCK

// ---- DUTs/Hardware/Insertion Package/Drives/ServoNC.TcPOU
FUNCTION_BLOCK ServoNC EXTENDS FBA_TrifectaDrive IMPLEMENTS I_EncodedDrive
VAR_OUTPUT	
	ready : BOOL;
	position : LREAL;
	velocity : LREAL;
END_VAR
VAR
	axis : AXIS_REF;
	
	mcReadPosition : MC_ReadActualPosition; //continuous enable FBs
	mcReadVelocity : MC_ReadActualVelocity;
	mcReadError : MC_ReadAxisError;
	mcPower : MC_Power;
	
	mcReset : MC_Reset; //rising edge FBs
	mcMoveAbsolute : MC_MoveAbsolute;
	mcMoveRelative : MC_MoveRelative;
	mcMoveVelocity : MC_MoveVelocity;
	
	mcSetPosition : MC_SetPosition;
	mcStop : MC_Stop;
END_VAR
VAR_STAT CONSTANT
	targetingVelocity : INT := 500;
	continuousVelocity : INT := 100;
END_VAR

override();

blocks();

mcReset.Execute := FALSE;
mcMoveAbsolute.Execute := FALSE;
mcMoveRelative.Execute := FALSE;
mcMoveVelocity.Execute := FALSE;
mcSetPosition.Execute := FALSE;
mcStop.Execute := FALSE;

blocks();

ready := bEnable AND NOT Active AND HomeSet;

PROPERTY Active : BOOL
GET
Active := 
	mcMoveAbsolute.Busy OR 
	mcMoveRelative.Busy OR 
	mcMoveVelocity.Busy OR 
	mcSetPosition.Busy OR 
	mcReset.Busy OR 
	mcStop.Busy OR 
	step <> 0;
END_GET
END_PROPERTY

METHOD PRIVATE blocks : BOOL
mcReadPosition(
	Axis:= axis, 
	Enable:= TRUE, 
	Valid=> , 
	Busy=> , 
	Error=> , 
	ErrorID=> , 
	Position=> position);
	
mcReadVelocity(
	Axis:= axis, 
	Enable:= TRUE, 
	Valid=> , 
	Busy=> , 
	Error=> , 
	ErrorID=> , 
	ActualVelocity=> velocity);
	
mcReadError(
	Axis:= axis, 
	Enable:= TRUE, 
	Valid=> , 
	Busy=> , 
	Error=> , 
	ErrorID=> , 
	AxisErrorID=> );

mcReset(
	Axis:= axis, 
	Execute:= , 
	Done=> , 
	Busy=> , 
	Error=> , 
	ErrorID=> );

mcPower(
	Axis:= axis, 
	Enable:= bEnable, 
	Enable_Positive:= TRUE, 
	Enable_Negative:= TRUE, 
	Override:= 100, 
	BufferMode:= , 
	Options:= , 
	Status=> , 
	Busy=> , 
	Active=> , 
	Error=> , 
	ErrorID=> );

mcMoveAbsolute(
	Axis:= axis, 
	Execute:= , 
	Position:= , 
	Velocity:= targetingVelocity, 
	Acceleration:= , 
	Deceleration:= , 
	Jerk:= , 
	BufferMode:= , 
	Options:= , 
	Done=> , 
	Busy=> , 
	Active=> , 
	CommandAborted=> , 
	Error=> , 
	ErrorID=> );
	
mcMoveRelative(
	Axis:= axis, 
	Execute:= , 
	Distance:= ,
	Velocity:= targetingVelocity, 
	Acceleration:= , 
	Deceleration:= , 
	Jerk:= , 
	BufferMode:= , 
	Options:= , 
	Done=> , 
	Busy=> , 
	Active=> , 
	CommandAborted=> , 
	Error=> , 
	ErrorID=> );
	
mcMoveVelocity( //stopped with stop();
	Axis:= axis, 
	Execute:= , 
	Velocity:= continuousVelocity, 
	Acceleration:= , 
	Deceleration:= , 
	Jerk:= , 
	Direction:= , 
	BufferMode:= , 
	Options:= , 
	InVelocity=> , 
	Busy=> , 
	Active=> , 
	CommandAborted=> , 
	Error=> , 
	ErrorID=> );
	
mcSetPosition(
	Axis:= axis, 
	Execute:= , 
	Position:= , 
	Mode:= , 
	Options:= , 
	Done=> , 
	Busy=> , 
	Error=> , 
	ErrorID=> );
	
mcStop(
	Axis:= axis, 
	Execute:= , 
	Deceleration:= , 
	Jerk:= , 
	Options:= , 
	Done=> , 
	Busy=> , 
	Active=> , 
	CommandAborted=> , 
	Error=> , 
	ErrorID=> );
END_METHOD

PROPERTY CurrentPosition : LREAL
GET
CurrentPosition := position;
END_GET
SET
position := CurrentPosition;
END_SET
END_PROPERTY

PROPERTY Error : BOOL
GET
error := 
	mcMoveAbsolute.Error OR 
	mcMoveRelative.Error OR 
	mcMoveVelocity.Error OR 
	mcSetPosition.Error OR 
	mcReset.Error OR 
	mcStop.Error OR
	mcReadError.AxisErrorID > 0;
END_GET
END_PROPERTY

METHOD homingSequence : BOOL
CASE step OF
	Homing.IDLE:
		reset();
		IF bEnable THEN
			step := Homing.START;
		END_IF
		
	Homing.START:
		IF AtHome THEN
			mcMoveVelocity.Execute := FALSE;
			step := Homing.STOP;
			
		ELSIF AtInnerLimit THEN
			mcMoveVelocity.Execute := FALSE;
			step := Homing.RETRY;
			
		ELSE
			mcMoveVelocity.Direction := MC_Negative_Direction;
			mcMoveVelocity.Execute := NOT mcMoveVelocity.Execute;
		END_IF
		
	Homing.RETRY:
		IF AtOuterLimit THEN
			mcMoveVelocity.Execute := FALSE;
			step := Homing.START;
		ELSE
			mcMoveVelocity.Direction := MC_Positive_Direction;
			mcMoveVelocity.Execute := NOT mcMoveVelocity.Execute;
		END_IF
		
	Homing.STOP:
		IF velocity = 0 THEN
			mcStop.Execute := FALSE;
			step := Homing.SET;
		ELSE
			mcStop.Execute := TRUE;
		END_IF
		
	Homing.SET:
		IF position = 0 THEN
			mcSetPosition.Execute := FALSE;
			homingSequence := TRUE;
			step := Homing.DONE;
		ELSE
			mcSetPosition.Position := 0;
			mcSetPosition.Execute := TRUE;
		END_IF
		
	Homing.DONE:
		homingComplete := TRUE;
		step := Homing.IDLE;
		
END_CASE
END_METHOD

METHOD moveAbsolute : BOOL
VAR_INPUT
	newTarget : LREAL;
END_VAR
(*
VAR_OUTPUT
	fault : BOOL;
END_VAR
*)
IF NOT Active AND NOT error THEN
	mcMoveAbsolute.Position := newTarget;
	mcMoveAbsolute.Execute := TRUE;
END_IF

moveAbsolute := (*mcMoveAbsolute.Done AND mcMoveAbsolute.Active;*)
	position = newTarget;
END_METHOD

METHOD moveContinuous : BOOL
VAR_INPUT
	//direction : BOOL; //direction (F = inwards, T = outwards)
	direction : MC_Direction;
END_VAR
(*
IF mcMoveVelocity.Active THEN
	stop();
END_IF

IF NOT mcStop.Done THEN
	RETURN;
END_IF
*)
(*
IF direction THEN
	mcMoveVelocity.Direction := MC_Positive_Direction;
ELSE
	mcMoveVelocity.Direction := MC_Negative_Direction;
END_IF
*)
mcMoveVelocity.Direction := direction;

IF NOT mcMoveVelocity.Error THEN
	mcMoveVelocity.Execute := TRUE;
	moveContinuous := TRUE;
END_IF
END_METHOD

METHOD moveRelative : BOOL
VAR_INPUT
	distance : LREAL;
END_VAR
mcMoveRelative.Distance := distance;

moveRelative := mcMoveRelative.Done;
END_METHOD

METHOD PRIVATE override : BOOL
VAR_INPUT
END_VAR
(*
-at home and attempting to traverse outward
-at outer limit and attempting to traverse outward
-at inner limit and attempting to traverse inwards
*)
(*
inward = negative direction, negative velocity
outward = positive direction, positive velocity
*)

IF error THEN
	stop();
	reset();
	
ELSIF
	AtHome AND (TargetPosition > CurrentPosition OR velocity > 0) OR
	AtInnerLimit AND (TargetPosition > CurrentPosition OR velocity > 0) OR
	AtOuterLimit AND (TargetPosition < CurrentPosition OR velocity < 0)
THEN
	stop();
END_IF
END_METHOD

METHOD reset : BOOL
VAR_INPUT
END_VAR
mcReset.Execute := TRUE;

reset := mcReset.Done;
END_METHOD

METHOD stop : BOOL
VAR_INPUT
END_VAR
mcStop.Execute := TRUE;

mcMoveAbsolute.Execute := FALSE;
mcMoveRelative.Execute := FALSE;
mcMoveVelocity.Execute := FALSE;
END_METHOD

PROPERTY TargetPosition : LREAL
GET
END_GET
SET
moveAbsolute(newTarget := TargetPosition);
END_SET
END_PROPERTY

METHOD toHome : BOOL
VAR_INPUT
END_VAR
moveAbsolute(newTarget := 0);

toHome := AtHome;
END_METHOD

END_FUNCTION_BLOCK

// ---- DUTs/Hardware/Insertion Package/Prototypes/FBA_TrifectaDrive.TcPOU
FUNCTION_BLOCK ABSTRACT FBA_TrifectaDrive EXTENDS FBA_Drive
VAR
	outerLimit AT %I* : BOOL;
END_VAR
(*
this abstract FB adds a rear limit sensor to FBA_Drive
*)

{attribute 'monitoring':='call'}
PROPERTY AtOuterLimit : BOOL
GET
AtOuterLimit := outerLimit <> limitSensorDefaultState;
END_GET
END_PROPERTY

END_FUNCTION_BLOCK

// ---- Sections/A22 - Cardboard/CardboardEx.TcPOU
FUNCTION_BLOCK CardboardEx EXTENDS SectionEx
VAR_IN_OUT
	benderLeft : FoldingMachine;
	
	robotLeft, robotRight : RobotA22;
	
	skidLeft, skidRight : SkidMagazine;
	magazineLeft, magazineRight : SkidMagazine;
	
	wrapper : WrapMachine;
	
	insertionLeft, insertionRight : Insertion;
	pistonBottom : SimplePiston;
	
	suctionTopLeft : ARRAY[*] OF SuctionPad; (*1..3*)
	suctionTopRight : ARRAY[*] OF SuctionPad; (*1..3*)
	suctionBottomLeft : ARRAY[*] OF SuctionPad; (*1..3*)
	suctionBottomRight : ARRAY[*] OF SuctionPad; (*1..3*)
	
	suctionBottom : ARRAY[*] OF SuctionPad; (*1..2*)
END_VAR
VAR	
	step : (IDLE, LOAD_SIDES_CORNERS, LOAD_TOP_BOTTOM, PUSH, TARGET_WRAP_POSITION, WRAP_AND_RELEASE, COMPLETE := 1050);
	
	masterLoadStep : INT;
	loadStepLeft, loadStepRight : INT;
	
	iWrap : INT;
	wrapPoints : INT;
	wrapRotations : INT;
	masterLength : INT;
	
	releaseDelayTimer : TON;
END_VAR
VAR //local types
	topLeftFoldsArr, topRightFoldsArr, bottomLeftFoldsArr, bottomRightFoldsArr : ARRAY[0..CONSTS.maxPairs] OF INT;
	
	//materialsArr : ARRAY[0..Consts.maxPairs] OF PositionMaterials;
	materialsArr : ARRAY[0..2*Consts.maxPairs] OF PositionMaterials;
	
	recipesCombined : BOOL;
	
	demoHeight : REAL := 640; //mm
	
	innerLoadedMaterials, outerLoadedMaterials : ARRAY[Surface.TOP..Surface.BOTTOM_RIGHT] OF STRING;
	//inner: cardboard by default
	//outer: corner guard by default
END_VAR
VAR CONSTANT
	releaseDelay : TIME := T#2000MS;
END_VAR
VAR
	//AOIs encapsulate functionality and reduce the number of module variables
	aoiCornerGuardLeft, aoiCornerGuardRight : AOI_LoadCornerGuard;
	aoiCornerCardboardLeft, aoiCornerCardboardRight : AOI_LoadCornerCardboard;
	aoiFlatCardboardLeft, aoiFlatCardboardRight : AOI_LoadFlatCardboard;
	
	//for testing only
	latchLeft, latchRight : BOOL; //prevents sliders from overshooting the inner limit sensor
	suctionEnableTopLeft, suctionEnableTopRight, suctionEnableBottomLeft, suctionEnableBottomRight : BOOL;
END_VAR

aoiBlocks();

SUPER^();

METHOD PROTECTED aoiBlocks : BOOL
VAR_INPUT
END_VAR
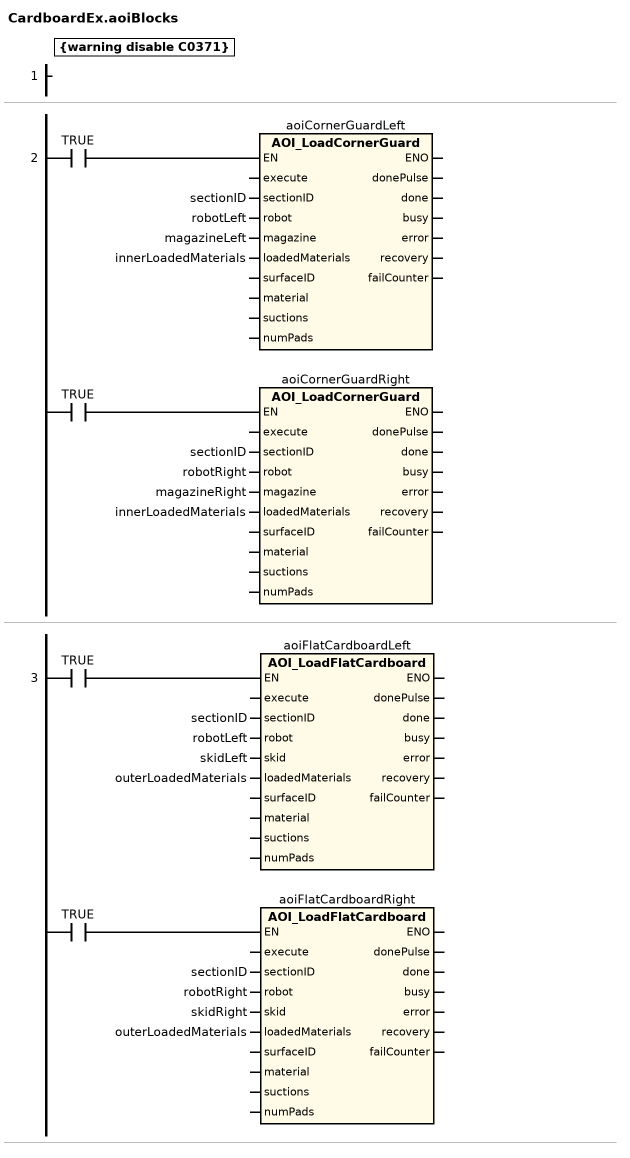
// NETWORK 1
// label: {warning disable C0371}

// NETWORK 2
aoiCornerGuardLeft(
    sectionID := sectionID,
    robot := robotLeft,
    magazine := magazineLeft,
    loadedMaterials := innerLoadedMaterials); // AOI_LoadCornerGuard
aoiCornerGuardRight(
    sectionID := sectionID,
    robot := robotRight,
    magazine := magazineRight,
    loadedMaterials := innerLoadedMaterials); // AOI_LoadCornerGuard

// NETWORK 3
aoiFlatCardboardLeft(
    sectionID := sectionID,
    robot := robotLeft,
    skid := skidLeft,
    loadedMaterials := outerLoadedMaterials); // AOI_LoadFlatCardboard
aoiFlatCardboardRight(
    sectionID := sectionID,
    robot := robotRight,
    skid := skidRight,
    loadedMaterials := outerLoadedMaterials); // AOI_LoadFlatCardboard
END_METHOD

METHOD PROTECTED combine : BOOL
VAR_IN_OUT
	cardboard : ARRAY[*] OF PositionMaterials;
	cornerGuard : ARRAY[*] OF PositionMaterials;
	
	combined : ARRAY[*] OF PositionMaterials;
END_VAR
VAR_INPUT
	cardboard_over_cornerGuard : BOOL;
END_VAR
VAR_INST
	topLength : REAL;
	leftLength : REAL;
	rightLength : REAL;
	bottomLength : REAL;
	
	topLeftLength : REAL;
	topRightLength : REAL;
	bottomLeftLength : REAL;
	bottomRightLength : REAL;
	
	outerMaterialLength : REAL;
	innerMaterialLength : REAL;
	
	i : INT;
	iCardboard : INT;
	iCornerGuard : INT;
END_VAR
FOR i:=0 TO CONSTS.maxPairs*2 BY 1 DO
	IF //no more cardboard (reached end of array or unused entries), 
		(iCardboard >= CONSTS.maxPairs OR_ELSE NOT PositionIsValid(cardboard[iCardboard])) AND_THEN //no more valid cardboard entries
		iCornerGuard < CONSTS.maxPairs AND_THEN //still has remaining corner guard
		PositionIsValid(cornerGuard[iCornerGuard]) //remaining corner guard is valid		
	THEN //finish with cornerguard
		combined[i] := cornerGuard[iCornerGuard];
		iCornerGuard := iCornerGuard + 1;
		CONTINUE;
	END_IF
	
	IF //no more cornerguard (reached end of array or unused entries)
		(iCornerGuard >= CONSTS.maxPairs OR_ELSE NOT PositionIsValid(cornerGuard[iCornerGuard])) AND_THEN
		iCardboard < CONSTS.maxPairs AND_THEN
		PositionIsValid(cardboard[iCardboard])
	THEN //finish with cardboard
		combined[i] := cardboard[iCardboard];
		iCardboard := iCardboard + 1;
		CONTINUE;
	END_IF
	
	(*
	IF NOT cardboard_over_cornerGuard THEN //cardboard on inside
		setOrder(cardboard, cornerGuard, combined, iCardboard, iCornerGuard, i);
		
	ELSE //cardboard on outside
		setOrder(cornerGuard, cardboard, combined, iCornerGuard, iCardboard, i);
		
	END_IF
	*)
END_FOR

combine := TRUE;
END_METHOD

METHOD PROTECTED load : BOOL
VAR_INPUT
	pairIndex : INT;
END_VAR
VAR_OUTPUT
	error : BOOL;
END_VAR
VAR
	pair : REFERENCE TO PositionMaterials REF= materialsArr[pairIndex];
	nextPair : REFERENCE TO PositionMaterials;
END_VAR
(*
unlike other sections, the load() function for cardboard + corner guard only loads the corners
to load flat cardboards, use the function loadFlats()
*)
{warning disable C0371}

IF robotLeft.error OR robotRight.error THEN
	RETURN;
ELSIF NOT (robotLeft.reserve(sectionID) AND robotRight.reserve(sectionID)) THEN //both robots must be reserved first
	RETURN;
END_IF

IF pairIndex + 1 < CONSTS.maxPairs THEN
	nextPair REF= materialsArr[pairIndex + 1];
END_IF

CASE masterLoadStep OF
	0: //check if next pair (which is to be placed over this pair) has the same position as this pair
		IF pairIndex + 1 >= CONSTS.maxPairs THEN //no next pair - NOTE: final pair is index 15 (16-1), not 16
			masterLoadStep := 10;
			loadStepLeft := loadStepRight := 0;
			
		ELSIF pair.position < nextPair.position THEN
			masterLoadStep := 10;
			loadStepLeft := loadStepRight := 0;
		(*	
		ELSIF MatchesMaterialType(pair:= nextPair, materialType:= 'CAR') AND_THEN loadCornerCardboards(pairIndex:= pairIndex + 1) THEN
			masterLoadStep := 10;
			loadStepLeft := loadStepRight := 0;
		*)
		ELSIF MatchesMaterialType(pair:= nextPair, materialPrefix:= 'COR') AND_THEN loadCornerGuards(pairIndex:= pairIndex + 1) THEN
			masterLoadStep := 10;
			loadStepLeft := loadStepRight := 0;
			
		END_IF
		
	10: //load this pair's side cardboards
		IF
			loadFlatCardboardsEx(
				robot:= robotLeft, 
				aoiLoad:= aoiFlatCardboardLeft, 
				loadStep:= loadStepLeft, 
				pairIndex:= pairIndex, 
				includeTop:= FALSE, 
				includeLeft:= TRUE, 
				includeRight:= FALSE, 
				includeBottom:= FALSE, 
				error=> )
			AND
			loadFlatCardboardsEx(
				robot:= robotLeft, 
				aoiLoad:= aoiFlatCardboardLeft, 
				loadStep:= loadStepLeft, 
				pairIndex:= pairIndex, 
				includeTop:= FALSE, 
				includeLeft:= FALSE, 
				includeRight:= TRUE, 
				includeBottom:= FALSE, 
				error=> )
		THEN
			masterLoadStep := 20;
			loadStepLeft := loadStepRight := 0;
		END_IF
		
	20: //load current pair
		IF
			MatchesMaterialType(pair:= pair, materialPrefix:= 'CAR') AND_THEN loadCornerCardboards(pairIndex:= iPair) OR_ELSE
			MatchesMaterialType(pair:= pair, materialPrefix:= 'COR') AND_THEN loadCornerGuards(pairIndex:= iPair)
		THEN //is cardboard
			loadStepLeft := loadStepRight := 0;
			masterLoadStep := COMPLETE;
		END_IF
	
	COMPLETE:
		robotLeft.release(sectionID);
		robotRight.release(sectionID);
		
		loadStepLeft := loadStepRight := 0;
		masterLoadStep := 0;
		load := TRUE;
	
END_CASE
END_METHOD

METHOD PROTECTED loadCornerCardboards : BOOL
VAR_INPUT
	pairIndex : INT;
END_VAR
VAR_OUTPUT
	error : BOOL;
END_VAR
VAR
	errorLeft, errorRight : BOOL;
	leftSuctionArr, rightSuctionArr : POINTER TO SuctionPad;
	leftNextSet, rightNextSet : INT;
	leftMaterial, rightMaterial : STRING;
	leftFold, rightFold : INT;
	
	pair : REFERENCE TO PositionMaterials REF= materialsArr[pairIndex];
	topLeftFold : INT := topLeftFoldsArr[pairIndex];
	topRightFold : INT := topRightFoldsArr[pairIndex];
	bottomLeftFold : INT := bottomLeftFoldsArr[pairIndex];
	bottomRightFold : INT := bottomRightFoldsArr[pairIndex];
END_VAR
{warning disable C0371}

loadCornerCardboards := 
	loadCornerCardboardsEx(
		robot:= robotLeft, 
		aoiLoad:= aoiCornerCardboardLeft, 
		loadStep:= loadStepLeft, 
		pairIndex:= pairIndex, 
		includeTopLeft:= TRUE, 
		includeTopRight:= FALSE, 
		includeBottomLeft:= TRUE, 
		includeBottomRight:= FALSE, 
		error=> errorLeft)
	AND
	loadCornerCardboardsEx(
		robot:= robotRight, 
		aoiLoad:= aoiCornerCardboardRight, 
		loadStep:= loadStepRight, 
		pairIndex:= pairIndex, 
		includeTopLeft:= FALSE, 
		includeTopRight:= TRUE, 
		includeBottomLeft:= FALSE, 
		includeBottomRight:= TRUE, 
		error=> errorLeft);
		
error := errorLeft OR errorRight;

(*
CASE cornerSetLeft OF
	0:
		leftNextSet := Surface.TOP_RIGHT;
		cornerSetLeft := 0;
		
	Surface.TOP_RIGHT: 
		leftNextSet := Surface.TOP_LEFT;
		leftSuctionArr := suctionTopRight;
		leftMaterial := pair.topRight;
		leftFold := topRightFold;
		
	Surface.TOP_LEFT: 
		leftNextSet := Surface.BOTTOM_RIGHT;
		leftSuctionArr := suctionTopLeft;
		leftMaterial := pair.topLeft;
		leftFold := topLeftFold;
		
	Surface.BOTTOM_RIGHT:
		leftNextSet := Surface.BOTTOM_LEFT;
		leftSuctionArr := suctionBottomRight;
		leftMaterial := pair.bottomRight;
		leftFold := bottomRightFold;
		
	Surface.BOTTOM_LEFT: 
		leftNextSet := COMPLETE;
		leftSuctionArr := suctionBottomLeft;
		leftMaterial := pair.bottomLeft;
		leftFold := bottomLeftFold;
END_CASE
IF
	(cornerSetLeft = 0 OR cornerSetLeft = COMPLETE) OR_ELSE
	leftCornerSequence(
		robot:= robotLeft, 
		skid:= skidLeft, 
		suctions := leftSuctionArr,
		loadStep:= loadStepLeft, 
		surfaceID:= cornerSetLeft,
		material:= pair.topRight, 
		foldPos0:= topRightFold, 
		foldPos1:= 0, 
		error=> )
THEN
	cornerSetLeft := leftNextSet;
	loadStepLeft := 0;
END_IF


CASE cornerSetRight OF
	0:
		cornerSetRight := Surface.TOP_RIGHT;
		rightSuctionArr := suctionTopRight;
		
	Surface.TOP_RIGHT:		
		rightNextSet := Surface.BOTTOM_RIGHT;
		rightSuctionArr := suctionTopRight;
		rightMaterial := pair.topRight;
		rightFold := topRightFold;
		
	Surface.BOTTOM_RIGHT: 
		rightNextSet := COMPLETE;
		rightSuctionArr := suctionBottomRight;
		rightMaterial := pair.bottomRight;
		rightFold := bottomRightFold;		
END_CASE
IF
	(cornerSetRight = 0 OR cornerSetRight = COMPLETE) OR_ELSE
	rightCornerSequence(
		robot:= robotRight, 
		skid:= skidRight, 
		suctions := rightSuctionArr,
		loadStep:= loadStepRight, 
		material:= pair.topRight, 
		surfaceID:= cornerSetRight,
		foldPos0:= pair.topRightFold, 
		foldPos1:= 0, 
		error=> )
THEN
	cornerSetRight := rightNextSet;
	loadStepRight := 0;
END_IF



IF cornerSetLeft = COMPLETE AND cornerSetRight = COMPLETE THEN
	loadCornerCardboards := TRUE;
	
	loadStepLeft := loadStepRight := 0;
	cornerSetLeft := cornerSetRight := 0;
END_IF
*)
END_METHOD

METHOD PROTECTED loadCornerCardboardsEx : BOOL
VAR_IN_OUT
	robot : RobotA22;
	aoiLoad : AOI_LoadCornerCardboard;
	loadStep : INT;
END_VAR
VAR_INPUT
	pairIndex : INT;
	includeTopLeft, includeTopRight, includeBottomLeft, includeBottomRight : BOOL;
END_VAR
VAR_OUTPUT
	error : BOOL;
END_VAR
VAR
	suctionsArrLeft, suctionsArrRight : POINTER TO SuctionPad;
	nextSetLeft, nextSetRight : INT;

	pair : REFERENCE TO PositionMaterials REF= materialsArr[pairIndex];
	topLeftFold : INT := topLeftFoldsArr[pairIndex];
	topRightFold : INT := topRightFoldsArr[pairIndex];
	bottomLeftFold : INT := bottomLeftFoldsArr[pairIndex];
	bottomRightFold : INT := bottomRightFoldsArr[pairIndex];
END_VAR
{warning disable C0371}

IF robot.error THEN
	error := TRUE;
	RETURN;
ELSIF robot.reservation <> sectionID AND_THEN NOT robot.reserve(sectionID) THEN
	RETURN;
ELSIF robot.tool <> sectionID AND_THEN NOT robot.changeEOAT(targetTool := sectionID) THEN
	RETURN;
END_IF

error := aoiLoad.error;

CASE loadStep OF
	0:
		loadStep := Surface.BOTTOM_LEFT;
		
	Surface.BOTTOM_LEFT:
		IF NOT includeBottomLeft OR aoiLoad.donePulse THEN
			aoiLoad.execute := FALSE;
			aoiLoad.material := '';
			loadStep := Surface.BOTTOM_RIGHT;
			RETURN;
		END_IF
		
		aoiLoad.surfaceID := loadStep;
		aoiLoad.material := pair.bottomLeft;
		aoiLoad.suctions := suctionBottomLeft;
		aoiLoad.numPads := UPPER_BOUND(suctionBottomLeft, 1) - LOWER_BOUND(suctionBottomLeft, 1) + 1;
		
		aoiLoad.foldPos0 := bottomLeftFold;
		aoiLoad.foldPos1 := 0;
		
		aoiLoad.execute := NOT aoiLoad.busy;
		
	Surface.BOTTOM_RIGHT:
		IF NOT includeBottomRight OR aoiLoad.donePulse THEN
			aoiLoad.execute := FALSE;
			aoiLoad.material := '';
			loadStep := Surface.TOP_LEFT;
			RETURN;
		END_IF
		
		aoiLoad.surfaceID := loadStep;
		aoiLoad.material := pair.bottomRight;
		aoiLoad.suctions := suctionBottomRight;
		aoiLoad.numPads := UPPER_BOUND(suctionBottomRight, 1) - LOWER_BOUND(suctionBottomRight, 1) + 1;
		
		aoiLoad.foldPos0 := bottomRightFold;
		aoiLoad.foldPos1 := 0;
		
		aoiLoad.execute := NOT aoiLoad.busy;
	
	Surface.TOP_LEFT:		
		IF NOT includeTopLeft OR aoiLoad.donePulse THEN
			aoiLoad.execute := FALSE;
			aoiLoad.material := '';
			loadStep := Surface.TOP_RIGHT;
			RETURN;
		END_IF
		
		aoiLoad.surfaceID := loadStep;
		aoiLoad.material := pair.top;
		aoiLoad.suctions := suctionTopLeft;
		aoiLoad.numPads := UPPER_BOUND(suctionTopLeft, 1) - LOWER_BOUND(suctionTopLeft, 1) + 1;
		
		aoiLoad.foldPos0 := topLeftFold;
		aoiLoad.foldPos1 := 0;
		
		aoiLoad.execute := NOT aoiLoad.busy;
		
	Surface.TOP_RIGHT:
		IF NOT includeTopRight OR aoiLoad.donePulse THEN
			aoiLoad.execute := FALSE;
			aoiLoad.material := '';
			loadStep := COMPLETE;
			RETURN;
		END_IF
		
		aoiLoad.surfaceID := loadStep;
		aoiLoad.material := pair.topRight;
		aoiLoad.suctions := suctionTopRight;
		aoiLoad.numPads := UPPER_BOUND(suctionTopRight, 1) - LOWER_BOUND(suctionTopRight, 1) + 1;
		
		aoiLoad.foldPos0 := topRightFold;
		aoiLoad.foldPos1 := 0;
		
		aoiLoad.execute := NOT aoiLoad.busy;
		
	COMPLETE:				
		robot.release(sectionID);
		
		aoiLoad.material := '';
		aoiLoad.execute := FALSE;
		
		loadCornerCardboardsEx := TRUE;
END_CASE
END_METHOD

METHOD loadCornerGuards : BOOL
VAR_INPUT
	pairIndex : INT;
END_VAR
VAR_OUTPUT
	error : BOOL;
END_VAR
VAR
	pair : REFERENCE TO PositionMaterials REF= materialsArr[pairIndex];
	errorLeft, errorRight : BOOL;
END_VAR
{warning disable C0371}

loadCornerGuards := 
	loadCornerGuardsEx(
		robot:= robotLeft, 
		aoiLoad:= aoiCornerGuardLeft, 
		loadStep:= loadStepLeft, 
		pairIndex:= pairIndex, 
		includeTopLeft:= TRUE, 
		includeTopRight:= FALSE, 
		includeBottomLeft:= TRUE, 
		includeBottomRight:= FALSE, 
		error=> errorLeft) 
	AND
	loadCornerGuardsEx(
		robot:= robotRight, 
		aoiLoad:= aoiCornerGuardRight, 
		loadStep:= loadStepRight, 
		pairIndex:= pairIndex, 
		includeTopLeft:= FALSE, 
		includeTopRight:= TRUE, 
		includeBottomLeft:= FALSE, 
		includeBottomRight:= TRUE, 
		error=> errorRight);
		
error := errorLeft OR errorRight;

(*
IF robotLeft.error OR robotRight.error THEN
	error := TRUE;
	RETURN;
	
ELSIF 
	(robotLeft.reservation <> sectionID AND_THEN NOT robotLeft.reserve(sectionID)) OR 
	(robotRight.reservation <> sectionID AND_THEN NOT robotRight.reserve(sectionID))
THEN //loading requires both robots be reserved together
	RETURN;
	
ELSIF //robots have wrong tool
	(robotLeft.tool <> sectionID AND_THEN NOT robotLeft.changeEOAT(targetTool := sectionID)) OR
	(robotRight.tool <> sectionID AND_THEN NOT robotRight.changeEOAT(targetTool := sectionID))
THEN
	RETURN;
	
END_IF

CASE loadStep OF
	0: //top and bottom
		IF aoiCornerGuardLeft.done AND aoiCornerGuardRight.done THEN
			aoiCornerGuardLeft.execute := aoiCornerGuardRight.execute := FALSE;
			aoiCornerGuardLeft.material := aoiCornerGuardRight.material := '';
			loadStep := 10;
			RETURN;
		END_IF
		
		aoiCornerGuardLeft.suctions := 0;
		aoiCornerGuardLeft.surfaceID := Surface.TOP;
		aoiCornerGuardLeft.material := pair.top;
		aoiCornerGuardLeft.numPads := 0;
		
		aoiCornerGuardRight.suctions := suctionBottom;
		aoiCornerGuardRight.surfaceID := Surface.BOTTOM;
		aoiCornerGuardRight.material := pair.bottom;
		aoiCornerGuardRight.numPads := 0;
		
		aoiCornerGuardLeft.execute := NOT aoiCornerGuardLeft.done AND NOT aoiCornerGuardLeft.busy;
		aoiCornerGuardRight.execute := NOT aoiCornerGuardRight.done AND NOT aoiCornerGuardRight.busy;
		
	10: //sides
		IF aoiCornerGuardLeft.done AND aoiCornerGuardRight.done THEN
			aoiCornerGuardLeft.execute := aoiCornerGuardRight.execute := FALSE;
			aoiCornerGuardLeft.material := aoiCornerGuardRight.material := '';
			loadStep := 10;
			RETURN;
		END_IF
		
		aoiCornerGuardLeft.suctions := 0;
		aoiCornerGuardLeft.surfaceID := Surface.LEFT;
		aoiCornerGuardLeft.material := pair.left;
		aoiCornerGuardLeft.numPads := 0;
		
		aoiCornerGuardRight.suctions := 0;
		aoiCornerGuardRight.surfaceID := Surface.RIGHT;
		aoiCornerGuardRight.material := pair.right;
		aoiCornerGuardRight.numPads := 0;
		
		aoiCornerGuardLeft.execute := NOT aoiCornerGuardLeft.done AND NOT aoiCornerGuardLeft.busy;
		aoiCornerGuardRight.execute := NOT aoiCornerGuardRight.done AND NOT aoiCornerGuardRight.busy;
		
	COMPLETE:
		loadStep := 0;
		loadCornerGuards := TRUE;
END_CASE

error := aoiCornerGuardLeft.error OR aoiCornerGuardRight.error;
*)
END_METHOD

METHOD loadCornerGuardsEx : BOOL
VAR_IN_OUT
	robot : RobotA22;
	aoiLoad : AOI_LoadCornerGuard;
	loadStep : INT;
END_VAR
VAR_INPUT
	pairIndex : INT;
	includeTopLeft, includeTopRight, includeBottomLeft, includeBottomRight : BOOL;
END_VAR
VAR_OUTPUT
	error : BOOL;
END_VAR
VAR
	pair : REFERENCE TO PositionMaterials REF= materialsArr[pairIndex];
END_VAR
{warning disable C0371}
IF robot.error THEN
	error := TRUE;
	RETURN;
ELSIF robot.reservation <> sectionID AND_THEN NOT robot.reserve(sectionID) THEN
	RETURN;
ELSIF robot.tool <> sectionID AND_THEN NOT robot.changeEOAT(targetTool := sectionID) THEN
	RETURN;
END_IF

error := aoiLoad.error;

CASE loadStep OF
	0:
		loadStep := Surface.BOTTOM_LEFT;
		
	Surface.BOTTOM_LEFT:
		IF NOT includeBottomLeft OR aoiLoad.donePulse THEN
			aoiLoad.execute := FALSE;
			aoiLoad.material := '';
			loadStep := Surface.BOTTOM_RIGHT;
			RETURN;
		END_IF
		
		aoiLoad.surfaceID := loadStep;
		aoiLoad.material := pair.bottomLeft;
		aoiLoad.suctions := suctionBottomLeft;
		aoiLoad.numPads := UPPER_BOUND(suctionBottomLeft, 1) - LOWER_BOUND(suctionBottomLeft, 1) + 1;
		
		aoiLoad.execute := NOT aoiLoad.busy;
		
	Surface.BOTTOM_RIGHT:
		IF NOT includeBottomRight OR aoiLoad.donePulse THEN
			aoiLoad.execute := FALSE;
			aoiLoad.material := '';
			loadStep := Surface.TOP_LEFT;
			RETURN;
		END_IF
		
		aoiLoad.surfaceID := loadStep;
		aoiLoad.material := pair.bottomRight;
		aoiLoad.suctions := suctionBottomRight;
		aoiLoad.numPads := UPPER_BOUND(suctionBottomRight, 1) - LOWER_BOUND(suctionBottomRight, 1) + 1;
		
		aoiLoad.execute := NOT aoiLoad.busy;
	
	Surface.TOP_LEFT:		
		IF NOT includeTopLeft OR aoiLoad.donePulse THEN
			aoiLoad.execute := FALSE;
			aoiLoad.material := '';
			loadStep := Surface.TOP_RIGHT;
			RETURN;
		END_IF
		
		aoiLoad.surfaceID := loadStep;
		aoiLoad.material := pair.top;
		aoiLoad.suctions := suctionTopLeft;
		aoiLoad.numPads := UPPER_BOUND(suctionTopLeft, 1) - LOWER_BOUND(suctionTopLeft, 1) + 1;
		
		aoiLoad.execute := NOT aoiLoad.busy;
		
	Surface.TOP_RIGHT:
		IF NOT includeTopRight OR aoiLoad.donePulse THEN
			aoiLoad.execute := FALSE;
			aoiLoad.material := '';
			loadStep := COMPLETE;
			RETURN;
		END_IF
		
		aoiLoad.surfaceID := loadStep;
		aoiLoad.material := pair.topRight;
		aoiLoad.suctions := suctionTopRight;
		aoiLoad.numPads := UPPER_BOUND(suctionTopRight, 1) - LOWER_BOUND(suctionTopRight, 1) + 1;
		
		aoiLoad.execute := NOT aoiLoad.busy;
		
	COMPLETE:				
		robot.release(sectionID);
		
		aoiLoad.material := '';
		aoiLoad.execute := FALSE;
		
		loadCornerGuardsEx := TRUE;
END_CASE
END_METHOD

METHOD PROTECTED loadFlatCardboards : BOOL
VAR_INPUT
	pairIndex : INT;
END_VAR
VAR_OUTPUT
	error : BOOL;
END_VAR
VAR
	pair : REFERENCE TO PositionMaterials REF= materialsArr[pairIndex];
	errorLeft, errorRight : BOOL;
END_VAR
{warning disable C0371}

loadFlatCardboards := 
	loadFlatCardboardsEx(
		robot:= robotLeft, 
		aoiLoad:= aoiFlatCardboardLeft, 
		loadStep:= loadStepLeft, 
		pairIndex:= pairIndex, 
		includeTop:= TRUE, 
		includeLeft:= FALSE, //left already loaded before
		includeRight:= FALSE, 
		includeBottom:= FALSE, 
		error=> errorLeft)
	AND
	loadFlatCardboardsEx(
		robot:= robotRight, 
		aoiLoad:= aoiFlatCardboardRight, 
		loadStep:= loadStepRight, 
		pairIndex:= pairIndex, 
		includeTop:= FALSE, 
		includeLeft:= FALSE, 
		includeRight:= FALSE, //right already loaded before
		includeBottom:= TRUE, 
		error=> errorRight);
		
error := errorLeft OR errorRight;

(*
IF robotLeft.error OR robotRight.error THEN
	error := TRUE;
	RETURN;
	
ELSIF 
	(robotLeft.reservation <> sectionID AND_THEN NOT robotLeft.reserve(sectionID)) OR 
	(robotRight.reservation <> sectionID AND_THEN NOT robotRight.reserve(sectionID))
THEN //loading requires both robots be reserved together
	RETURN;
	
ELSIF //robots have wrong tool
	(robotLeft.tool <> sectionID AND_THEN NOT robotLeft.changeEOAT(targetTool := sectionID)) OR
	(robotRight.tool <> sectionID AND_THEN NOT robotRight.changeEOAT(targetTool := sectionID))
THEN
	RETURN;
	
END_IF

CASE loadStep OF
	0: //top and bottom
		IF aoiFlatCardboardLeft.done AND aoiFlatCardboardRight.done THEN
			aoiFlatCardboardLeft.execute := aoiFlatCardboardRight.execute := FALSE;
			aoiFlatCardboardLeft.material := aoiFlatCardboardRight.material := '';
			loadStep := 10;
			RETURN;
		END_IF
		
		aoiFlatCardboardLeft.suctions := 0;
		aoiFlatCardboardLeft.surfaceID := Surface.TOP;
		aoiFlatCardboardLeft.material := pair.top;
		aoiFlatCardboardLeft.numPads := 0;
		
		aoiFlatCardboardRight.suctions := suctionBottom;
		aoiFlatCardboardRight.surfaceID := Surface.BOTTOM;
		aoiFlatCardboardRight.material := pair.bottom;
		aoiFlatCardboardRight.numPads := 0;
		
		aoiFlatCardboardLeft.execute := NOT aoiFlatCardboardLeft.done AND NOT aoiFlatCardboardLeft.busy;
		aoiFlatCardboardRight.execute := NOT aoiFlatCardboardRight.done AND NOT aoiFlatCardboardRight.busy;
		
	10: //sides
		IF aoiFlatCardboardLeft.done AND aoiFlatCardboardRight.done THEN
			aoiFlatCardboardLeft.execute := aoiFlatCardboardRight.execute := FALSE;
			aoiFlatCardboardLeft.material := aoiFlatCardboardRight.material := '';
			loadStep := 10;
			RETURN;
		END_IF
		
		aoiFlatCardboardLeft.suctions := 0;
		aoiFlatCardboardLeft.surfaceID := Surface.LEFT;
		aoiFlatCardboardLeft.material := pair.left;
		aoiFlatCardboardLeft.numPads := 0;
		
		aoiFlatCardboardRight.suctions := 0;
		aoiFlatCardboardRight.surfaceID := Surface.RIGHT;
		aoiFlatCardboardRight.material := pair.right;
		aoiFlatCardboardRight.numPads := 0;
		
		aoiFlatCardboardLeft.execute := NOT aoiFlatCardboardLeft.done AND NOT aoiFlatCardboardLeft.busy;
		aoiFlatCardboardRight.execute := NOT aoiFlatCardboardRight.done AND NOT aoiFlatCardboardRight.busy;
		
	COMPLETE:
		loadStepLeft := loadStepRight := 0;
		loadStep := 0;
		
		loadFlatCardboards := TRUE;
END_CASE

error := aoiFlatCardboardLeft.error OR aoiFlatCardboardRight.error;
*)
END_METHOD

METHOD loadFlatCardboardsEx : BOOL
VAR_IN_OUT
	robot : RobotA22;
	aoiLoad : AOI_LoadFlatCardboard;
	loadStep : INT;
END_VAR
VAR_INPUT
	pairIndex : INT;
	includeTop, includeLeft, includeRight, includeBottom : BOOL;
END_VAR
VAR_OUTPUT
	error : BOOL;
END_VAR
VAR
	pair : REFERENCE TO PositionMaterials REF= materialsArr[pairIndex];
END_VAR
IF robot.error THEN
	error := TRUE;
	RETURN;
ELSIF robot.reservation <> sectionID AND_THEN NOT robot.reserve(sectionID) THEN
	RETURN;
ELSIF robot.tool <> sectionID AND_THEN NOT robot.changeEOAT(targetTool := sectionID) THEN
	RETURN;
END_IF

error := aoiLoad.error;

CASE loadStep OF
	0:
		loadStep := Surface.TOP;
	
	Surface.TOP:	
		IF NOT includeTop OR aoiLoad.donePulse THEN
			aoiLoad.execute := FALSE;
			aoiLoad.material := '';
			loadStep := Surface.BOTTOM;
			RETURN;
		END_IF
		
		aoiLoad.surfaceID := Surface.TOP;
		aoiLoad.material := pair.top;
		aoiLoad.suctions := 0;
		aoiLoad.numPads := 0;
		
		aoiLoad.execute := NOT aoiLoad.busy;
		
	Surface.BOTTOM:
		IF NOT includeBottom OR aoiLoad.donePulse THEN
			aoiLoad.execute := FALSE;
			aoiLoad.material := '';
			loadStep := Surface.LEFT;
			RETURN;
		END_IF
		
		aoiLoad.surfaceID := Surface.BOTTOM;
		aoiLoad.material := pair.bottom;
		aoiLoad.suctions := suctionBottom;
		aoiLoad.numPads := UPPER_BOUND(suctionBottom, 1) - LOWER_BOUND(suctionBottom, 1) + 1;
		
		aoiLoad.execute := NOT aoiLoad.busy;
		
	Surface.LEFT:
		IF NOT includeLeft OR aoiLoad.donePulse THEN
			aoiLoad.execute := FALSE;
			aoiLoad.material := '';
			loadStep := Surface.RIGHT;
			RETURN;
		END_IF
		
		aoiLoad.surfaceID := Surface.LEFT;
		aoiLoad.material := pair.left;
		aoiLoad.suctions := 0;
		aoiLoad.numPads := 0;
		
		aoiLoad.execute := NOT aoiLoad.busy;
		
	Surface.RIGHT:
		IF NOT includeRight OR aoiLoad.donePulse THEN
			aoiLoad.execute := FALSE;
			aoiLoad.material := '';
			loadStep := COMPLETE;
			RETURN;
		END_IF
		
		aoiLoad.surfaceID := Surface.RIGHT;
		aoiLoad.material := pair.right;
		aoiLoad.suctions := 0;
		aoiLoad.numPads := 0;
		
		aoiLoad.execute := NOT aoiLoad.busy;
		
	COMPLETE:				
		robot.release(sectionID);
		
		aoiLoad.material := '';
		aoiLoad.execute := FALSE;
		
		loadFlatCardboardsEx := TRUE;
END_CASE
END_METHOD

METHOD PROTECTED maintenance : BOOL
VAR_INPUT
END_VAR
{warning disable C0371}
IF robotLeft.Done THEN
	robotLeft.clearCommand();
END_IF

IF robotRight.Done THEN
	robotRight.clearCommand();
END_IF
END_METHOD

METHOD PROTECTED manual : BOOL
VAR_INPUT
END_VAR
END_METHOD

METHOD PROTECTED process : BOOL
VAR_INPUT
	auto : BOOL;
END_VAR
VAR_OUTPUT
	error : BOOL;
END_VAR
VAR
	currentPair : REFERENCE TO PositionMaterials REF= materialsArr[iPair];
END_VAR
{warning disable C0371}

IF iPair >= CONSTS.maxPairs THEN
	process := TRUE;
	RETURN;
ELSIF NOT PositionIsValid(pair := currentPair) THEN
	iPair := iPair + 1;
	RETURN;
END_IF
(*
corrected sequence:
	load sides
	load corners
	load bottom
	load top
*)

CASE step OF
	IDLE:
		IF trigger.Q THEN
			step := LOAD_SIDES_CORNERS;
		END_IF
	
	LOAD_SIDES_CORNERS: //load
		IF
			(auto AND done) OR
			(NOT auto AND trigger.Q)
		THEN
			aoiCornerCardboardLeft.reset();
			aoiCornerCardboardRight.reset();
			
			aoiCornerGuardLeft.reset();
			aoiCornerGuardRight.reset();
			
			aoiFlatCardboardLeft.reset();
			aoiFlatCardboardRight.reset();
			
			step := LOAD_TOP_BOTTOM;
			RETURN;
		END_IF
		
		IF NOT done THEN
			done := load(pairIndex := iPair);
		END_IF
		
	LOAD_TOP_BOTTOM:
		IF
			(auto AND done) OR
			(NOT auto AND trigger.Q)
		THEN
			aoiCornerCardboardLeft.reset();
			aoiCornerCardboardRight.reset();
			
			aoiCornerGuardLeft.reset();
			aoiCornerGuardRight.reset();
			
			aoiFlatCardboardLeft.reset();
			aoiFlatCardboardRight.reset();
			
			step := PUSH;
			RETURN;
		END_IF
		
		IF NOT done THEN
			done := loadFlatCardboards(pairIndex := iPair);
		END_IF
		
	PUSH:
		IF
			(auto AND latchLeft AND latchRight AND pistonBottom.extended) OR
			(NOT auto AND trigger.Q)
		THEN
			step := TARGET_WRAP_POSITION;
			RETURN;
		END_IF
		
		insertionLeft.align(demoHeight+5);
		insertionRight.align(demoHeight+5);
		
		IF //align slider to 5mm gap above bundle height
			insertionLeft.sliderPos <> demoHeight+5 OR
			insertionRight.sliderPos <> demoHeight+5
		THEN
			RETURN;
		END_IF
		
		IF NOT latchLeft THEN
			latchLeft := insertionLeft.contact;
			insertionLeft.press();
		END_IF
		
		IF NOT latchRight THEN
			latchRight := insertionRight.contact;
			insertionRight.press();
		END_IF
		
		pistonBottom.extend();
		
	TARGET_WRAP_POSITION:		
		IF iWrap >= wrapPoints THEN
			step := COMPLETE;
			RETURN;
		END_IF
		
		IF materialsArr[iPair].position = materialsArr[iPair + 1].position THEN //if this and the next pair were loaded together
			masterLength := TO_INT( MAX( GetPairMasterLength(materialsArr[iPair]), GetPairMasterLength(materialsArr[iPair + 1]) ) );
			wrapPoints := MAX( materialsArr[iPair].wrapPoints, materialsArr[iPair + 1].wrapPoints );
			wrapRotations := MAX( materialsArr[iPair].wrapRotations, materialsArr[iPair + 1].wrapRotations );
		ELSE
			masterLength := TO_INT( GetPairMasterLength(materialsArr[iPair]) );
			wrapPoints := materialsArr[iPair].wrapPoints;
			wrapRotations := materialsArr[iPair].wrapRotations;
		END_IF
		
		(*
		directionCheckAndSet(
			wrapConveyorPos,
			(currentPair.position - masterLength/2) + (masterLength/(currentPair.wrapPoints + 1) * (iWrap + 1)));
		*)
		step := WRAP_AND_RELEASE;
		
	WRAP_AND_RELEASE:
		releaseDelayTimer(IN:= , PT:= releaseDelay, Q=> , ET=> );
		
		IF wrapper.ready THEN
			wrapper.wrap(wrapRotations);
			releaseDelayTimer.IN := TRUE;
		END_IF
		
		IF releaseDelayTimer.Q THEN
			SetSuctions(suctions := suctionTopLeft, state := FALSE);
			SetSuctions(suctions := suctionTopRight, state := FALSE);
			SetSuctions(suctions := suctionBottomLeft, state := FALSE);
			SetSuctions(suctions := suctionBottomRight, state := FALSE);
			
			insertionLeft.toHome();
			insertionRight.toHome();
			pistonBottom.retract();
		END_IF
		
		IF wrapper.done AND insertionLeft.home AND insertionRight.home AND pistonBottom.retracted THEN
			releaseDelayTimer.IN := FALSE;
			step := WRAP_AND_RELEASE;
		END_IF
	
	COMPLETE:
		iPair := iPair + 1;
		iWrap := wrapPoints := wrapRotations := 0;
		step := IDLE;
		
END_CASE
END_METHOD

METHOD PROTECTED ps_AbortCondition : BOOL
VAR_INPUT
END_VAR
{warning disable C0371}
ps_AbortCondition :=
	insertionLeft.error OR 
	insertionRight.error OR 
	robotLeft.error OR 
	robotRight.error OR
	wrapper.error;
END_METHOD

METHOD PROTECTED ps_Aborted : BOOL
VAR_INPUT
END_VAR
ps_Aborted := TRUE;
END_METHOD

METHOD PROTECTED ps_Aborting : BOOL
VAR_INPUT
END_VAR
{warning disable C0371}
insertionLeft.stop();
insertionRight.stop();
pistonBottom.stop();

aoiFlatCardboardLeft.reset();
aoiFlatCardboardRight.reset();

aoiCornerCardboardLeft.reset();
aoiCornerCardboardRight.reset();

aoiCornerGuardLeft.reset();
aoiCornerGuardRight.reset();

robotLeft.clearCommand();
robotRight.clearCommand();

//stop conveyors

ps_Aborting :=
	NOT insertionLeft.active AND
	NOT insertionRight.active AND
	NOT pistonBottom.busy AND
	NOT robotLeft.Busy AND
	NOT robotRight.Busy;
END_METHOD

METHOD PROTECTED ps_Clearing : BOOL
VAR_INPUT
END_VAR
{warning disable C0371}
insertionLeft.reset();
insertionRight.reset();

ps_Clearing := 
	NOT insertionLeft.error AND
	NOT insertionRight.error AND
	NOT wrapper.error AND
	NOT robotLeft.error AND
	NOT robotRight.error;
END_METHOD

METHOD PROTECTED ps_Complete : BOOL
VAR_INPUT
END_VAR
ps_Complete := TRUE;
END_METHOD

METHOD PROTECTED ps_Completing : BOOL
VAR_INPUT
END_VAR
ps_Completing := NOT occupied;
END_METHOD

METHOD PROTECTED ps_Held : BOOL
VAR_INPUT
END_VAR
ps_Held := NOT hold;
END_METHOD

METHOD PROTECTED ps_HoldCondition : BOOL
VAR_INPUT
END_VAR
END_METHOD

METHOD PROTECTED ps_Holding : BOOL
VAR_INPUT
END_VAR
{warning disable C0371}
insertionLeft.stop();
insertionRight.stop();
pistonBottom.stop();
//set robot to pause

ps_Holding :=
	NOT insertionLeft.active AND
	NOT insertionRight.active;
END_METHOD

METHOD PROTECTED ps_Resetting : BOOL
VAR_INPUT
END_VAR
{warning disable C0371}
insertionLeft.reset();
insertionRight.reset();

ps_Resetting := 
	reset AND
	NOT insertionLeft.error AND
	NOT insertionRight.error AND
	NOT wrapper.error AND
	NOT robotLeft.error AND
	NOT robotRight.error;
END_METHOD

METHOD PROTECTED ps_Starting : BOOL
VAR_INPUT
END_VAR
{warning disable C0371}
robotLeft.clearCommand();
robotRight.clearCommand();

insertionLeft.homingSequence();
insertionRight.homingSequence();
pistonBottom.retract();

ps_Starting := 
	insertionLeft.screw.HomeSet AND 
	insertionRight.screw.HomeSet AND 
	pistonBottom.retracted;
END_METHOD

METHOD PROTECTED ps_StopCondition : BOOL
VAR_INPUT
END_VAR
ps_StopCondition := 
	stop;
END_METHOD

METHOD PROTECTED ps_Stopped : BOOL
VAR_INPUT
END_VAR
ps_Stopped := TRUE;
END_METHOD

METHOD PROTECTED ps_Stopping : BOOL
VAR_INPUT
END_VAR
{warning disable C0371}
insertionLeft.stop();
insertionRight.stop();
pistonBottom.stop();

aoiFlatCardboardLeft.reset();
aoiFlatCardboardRight.reset();

aoiCornerCardboardLeft.reset();
aoiCornerCardboardRight.reset();

aoiCornerGuardLeft.reset();
aoiCornerGuardRight.reset();

robotLeft.clearCommand();
robotRight.clearCommand();

wrapper.bEnable := FALSE;

//stop conveyors

ps_Stopping :=
	//NOT insertionLeft.active AND
	NOT insertionRight.active AND
	NOT pistonBottom.busy AND
	NOT robotLeft.Busy AND
	NOT robotRight.Busy AND
	NOT wrapper.busy;
END_METHOD

METHOD PROTECTED ps_SuspendCondition : BOOL
VAR_INPUT
END_VAR
END_METHOD

METHOD PROTECTED ps_Suspended : BOOL
VAR_INPUT
END_VAR
ps_Suspended := NOT ps_SuspendCondition();
END_METHOD

METHOD PROTECTED ps_Suspending : BOOL
VAR_INPUT
END_VAR
ps_Suspending := TRUE;
END_METHOD

METHOD PROTECTED ps_Unholding : BOOL
VAR_INPUT
END_VAR
ps_Unholding := TRUE;
END_METHOD

METHOD PROTECTED ps_Unsuspending : BOOL
VAR_INPUT
END_VAR
ps_Unsuspending := TRUE;
END_METHOD

METHOD PROTECTED runSectionTasks : BOOL
VAR_INPUT
	auto : BOOL;
END_VAR
VAR_OUTPUT
	error : BOOL;
END_VAR
SUPER^.runSectionTasks(auto := auto, error => error);

CASE status OF
	SectionTask.IDLE:
		RETURN;
	
	SectionTask.ALIGN:
		IF NOT recipesCombined THEN
			combine(
				currentBundle.cardboard, 
				currentBundle.cornerGuard, 
				materialsArr, 
				currentBundle.cardboard_over_cornerGuard);
				
			recipesCombined := TRUE;
		END_IF
		
	SectionTask.ACTIVE:
		recipesCombined := FALSE;
		
	SectionTask.DISCHARGE:
		//
		
	SectionTask.COMPLETE:	
		//
		
	-100:
		RETURN;
		
END_CASE
END_METHOD

METHOD PROTECTED setOrder : BOOL
VAR_IN_OUT
	innerArray : ARRAY[*] OF PositionMaterials;
	outerArray : ARRAY[*] OF PositionMaterials;
	
	combined : ARRAY[*] OF PositionMaterials;
	
	i_inner : INT;
	i_outer : INT;
	i_combined : INT;
END_VAR
VAR	
	outerMaterialLength : LREAL;
	innerMaterialLength : LREAL;
END_VAR
//if inner material is in front of outer material, inner material goes first
IF innerArray[i_inner].position <= outerArray[i_outer].position THEN

	combined[i_combined] := innerArray[i_inner];
	i_inner := i_inner + 1; //check next cardboard during next iteration
	
	setOrder := TRUE;
	RETURN;
END_IF
	
outerMaterialLength := GetPairMasterLength(outerArray[i_outer]);
innerMaterialLength := GetPairMasterLength(innerArray[i_inner]);

//if current inner material is too close to current outer material, place inner material first
//compare inner materials' front with outer material's back
IF (innerArray[i_inner].position - innerMaterialLength/2) < (outerArray[i_outer].position + outerMaterialLength/2) THEN
	combined[i_combined] := innerArray[i_inner];
	i_inner := i_inner + 1;
ELSE //otherwise, outer material can go
	combined[i_combined] := outerArray[i_outer];
	i_outer := i_outer + 1;
END_IF

setOrder := TRUE;
END_METHOD

METHOD PROTECTED unload : BOOL
VAR_INPUT
END_VAR
END_METHOD

END_FUNCTION_BLOCK

// ---- Sections/Abstract/SectionEx.TcPOU
FUNCTION_BLOCK ABSTRACT SectionEx
VAR_INPUT
	enable : BOOL;
	sectionID : SectionEnum;
END_VAR
VAR_IN_OUT
	bundlesQueue : ARRAY[*] OF Bundle;
	conveyorsArr : ARRAY[*] OF POINTER TO ConveyorSC;
	//in addition to the conveyos array, each section must receive references to the origial conveyors the array elements point to
END_VAR
VAR_OUTPUT
	activeBundle : Bundle; //assigned if there is a bundle to target
	bypass : BOOL; //assigned once the bundle head passes the section (status >= ACTIVE)
END_VAR
VAR_OUTPUT //PackML states + controls
	run : BOOL;
	stop : BOOL;
	hold : BOOL;
	reset : BOOL;
	
	ready : BOOL;
	busy : BOOL;
	done : BOOL;
	error : BOOL;
	
	pmlModeString : STRING;
	pmlStateString : STRING;
	
	pmlState : E_PMLState;
	pmlMode : E_PMLCustomUnitMode;
	
	iBundle : INT(0..Consts.maxQueue);
	iPair : INT(0..Consts.maxPairs);
END_VAR
VAR //PackML types
	pmlCommand : E_PMLCommand;
	pmlModeRequest : E_PMLCustomUnitMode := ePMLCustomUnitMode_Production;
	
	pmlStateMachine : PML_StateMachine;
	pmlModeManager : PML_UnitModeManager;
	pmlSemiAutoConfig : PML_UnitModeConfig;
END_VAR
VAR
	execute AT %M* : BOOL; //change to %I* depending on needs
	trigger : R_TRIG;
	
	currentBundle : REFERENCE TO Bundle;
	loadedMaterials : ARRAY[Surface.TOP..Surface.BOTTOM_RIGHT] OF STRING;

	requestedConveyorMode : ConveyorMode;
	conveyorPos : REAL;
	
	nextSection : POINTER TO SectionEx;
	prevSection : POINTER TO SectionEx;
	
	occupied : BOOL; //may be a dedicated sensor or a conveyor sensor
	
	status : SectionTask; //section status
END_VAR
VAR_STAT CONSTANT
	INCLUSIVE : INT := 0;
	EXCLUSIVE : INT := 1;
	COMPLETE : INT := 1030;
	
	suctionReleaseDelay : TIME := T#1000MS;
END_VAR

currentBundle REF= bundlesQueue[iBundle];
bypass := currentBundle.bypass;

ready := status = 0;
busy := status > 0;
done := done;
error := error;

blocks();
configPmlModes();

trigger(CLK:= execute, Q=> );

(*
PackML
	state machine for packaging applications - see Tc3_PackML_V2 library on InfoSys
	
	final states - wait for an input or condition and command to new state
	intermediate states - complete a task and call pmlStateMachine.M_StateComplete() to advance to next state
	
the following states currently use the same logic (albeit in different methods), implementation may change later
	ps_Stopping() and ps_Aborting()
	ps_Resetting() and ps_Clearing()
	
STOP - controlled stop **with intent to shutdown or vacate for extended time** induced by operator/HMI - otherwise use HOLD
ABORT - emergency stop due to machine errors

HOLD - minor local issues
SUSPEND - external issues

EXECUTE - major control logic
	different modes may require different tasks
	create methods as required for different modes, then call the correct method in ps_Completing()
	can be commanded to STOP, ABORT, HOLD, or SUSPEND at any point
COMPLETING - process complete, move product out of system and finish transition to COMPLETED

the implementation below can be copied to all POUs that use a PackML state machine
the individual ps_< > methods need to be implemented for the specific application
*)

IF ps_AbortCondition() THEN //abort condition
	pmlCommand := ePMLCommand_Abort;
ELSIF ps_StopCondition() THEN //stop condition
	pmlCommand := ePMLCommand_Stop;
END_IF

CASE pmlState OF
	0 (*ePMLState_Undefined*): //default state on startup
		pmlCommand := ePMLCommand_Stop;
		
	ePMLState_Stopping:
		IF ps_Stopping() THEN
			pmlStateMachine.M_StateComplete();
		END_IF
		
	ePMLState_Stopped:
		IF ps_Stopped() THEN
			pmlCommand := ePMLCommand_Reset;
		END_IF
	
    ePMLState_Resetting:
		IF ps_Resetting() THEN
			pmlStateMachine.M_StateComplete();
		END_IF
		
	ePMLState_Idle:
		IF ps_Idle() THEN
			pmlCommand := ePMLCommand_Start;
		END_IF		
	
	ePMLState_Starting:
		IF ps_Starting() THEN
			pmlStateMachine.M_StateComplete();
		END_IF
	
	ePMLState_Execute: //check the conditions in order of their priority, currently HOLD has the highest priority
		IF ps_HoldCondition() THEN
			pmlCommand := ePMLCommand_Hold;
			
		ELSIF ps_SuspendCondition() THEN
			pmlCommand := ePMLCommand_Suspend;			
		
		ELSIF ps_Execute(error => error) THEN //ps_Execute.error => THIS^.error
			pmlStateMachine.M_StateComplete();
			pmlCommand := ePMLCommand_Complete;
		END_IF
		
	ePMLState_Completing:
		IF ps_Completing() THEN
			pmlStateMachine.M_StateComplete();
		END_IF
	
	ePMLState_Complete:
		IF ps_Complete() THEN
			pmlCommand := ePMLCommand_Reset;
		END_IF
	
	ePMLState_Holding:
		IF ps_Holding() THEN
			pmlStateMachine.M_StateComplete();
		END_IF
	
	ePMLState_Held:
		IF NOT hold THEN
			pmlCommand := ePMLCommand_Unhold;
		END_IF
	
	ePMLState_Unholding:
		IF ps_Unholding() THEN
			pmlStateMachine.M_StateComplete(); //release all pause commands and IO
		END_IF
		
	ePMLState_Suspending: //based on next section conditions
		IF ps_Suspending() THEN
			pmlStateMachine.M_StateComplete();
		END_IF
		
	ePMLState_Suspended: //based on next section conditions
		IF ps_Suspended() THEN
			pmlCommand := ePMLCommand_Unsuspend;
		END_IF
	
	ePMLState_Unsuspending: //based on next section conditions
		IF ps_Unsuspending() THEN
			pmlStateMachine.M_StateComplete();
		END_IF
	
	ePMLState_Aborting:
		IF ps_Aborting() THEN
			pmlStateMachine.M_StateComplete();
		END_IF
	
	ePMLState_Aborted:
		IF ps_Aborted() THEN
			pmlCommand := ePMLCommand_Clear;
		END_IF
	
	ePMLState_Clearing:
		IF ps_Clearing() THEN
			pmlStateMachine.M_StateComplete();
		END_IF
	
END_CASE

METHOD PROTECTED blocks : BOOL
pmlModeManager(
	bExecute:= NOT pmlModeManager.bExecute, 
	eModeCommand:= pmlModeRequest, 
	eState:= pmlState, 
	eModeStatus=> pmlMode, 
	sModeStatus=> pmlModeString, 
	bDone=> , 
	bError=> , 
	nErrorId=> );

pmlStateMachine(
	eMode:= pmlMode, 
	eCommand:= pmlCommand, 
	stSubUnitInfoRef:= , 
	stOptions:= , 
	eState=> pmlState, 
	sState=> pmlStateString, 
	bError=> , 
	nErrorID=> );
END_METHOD

METHOD PROTECTED configPmlModes : BOOL
pmlSemiAutoConfig(
	eMode:= 4, 
	sName:= 'SemiAuto', 
	bDisableClearing:= FALSE, 
	bDisableStarting:= FALSE, 
	bDisableSuspended:= FALSE, 
	bDisableStopping:= FALSE, 
	bDisableAborting:= FALSE, 
	bDisableHolding:= FALSE, 
	bDisableHeld:= FALSE, 
	bDisableUnholding:= FALSE, 
	bDisableSuspending:= FALSE, 
	bDisableUnsuspending:= FALSE, 
	bDisableResetting:= FALSE, 
	bDisableIdle:= FALSE, 
	bDisableCompleting:= FALSE, 
	bDisableComplete:= FALSE, 
	bEnableUnitModeChangeStopped:= TRUE, 
	bEnableUnitModeChangeIdle:= TRUE, 
	bEnableUnitModeChangeSuspended:= FALSE, 
	bEnableUnitModeChangeExecute:= FALSE, 
	bEnableUnitModeChangeAborted:= TRUE, 
	bEnableUnitModeChangeHeld:= FALSE, 
	bEnableUnitModeChangeComplete:= FALSE, 
	bError=> , 
	nErrorId=> );
END_METHOD

METHOD connectTo : BOOL
VAR_INPUT
	connectedSection : POINTER TO SectionEx;
END_VAR
nextSection := connectedSection;

IF connectedSection <> 0 THEN
	connectedSection^.prevSection := THIS;
END_IF
END_METHOD

METHOD PROTECTED directionCheckAndSet : BOOL
VAR_INPUT
	conveyorRef : REAL;
	target : REAL;
END_VAR
//returns true conveyorRef is in range of target
IF WithinTolerance(value:= conveyorRef, target:= target, tolerance:= CONSTS.precisionTolerance) THEN
	directionCheckAndSet := TRUE;
	
ELSIF conveyorRef > target THEN
	pConveyorMode := ConveyorMode.BACKWARD;
	
ELSIF conveyorRef < target THEN
	pConveyorMode := ConveyorMode.FORWARD;
	
END_IF
END_METHOD

METHOD PROTECTED ABSTRACT load : BOOL
VAR_INPUT
	pairIndex : INT;
END_VAR
VAR_OUTPUT
	error : BOOL;
END_VAR
(*
loading takes place while the section is NOT active
materials are loaded for the next incoming bundle, not the current bundle - may differ for each section
*)
END_METHOD

METHOD PROTECTED ABSTRACT maintenance : BOOL
VAR_INPUT
END_VAR
END_METHOD

METHOD PROTECTED ABSTRACT manual : BOOL
VAR_INPUT
END_VAR
END_METHOD

PROPERTY PROTECTED pConveyorMode : ConveyorMode
GET
pConveyorMode := requestedConveyorMode;
END_GET
SET
VAR
	i : DINT;
END_VAR
requestedConveyorMode := pConveyorMode;

FOR i:=LOWER_BOUND(conveyorsArr, 1) TO UPPER_BOUND(conveyorsArr, 1) BY 1 DO
	
	CASE status OF
		SectionTask.ALIGN, -100:
			//all conveyors requested to same mode
			conveyorsArr[i]^.setRequest(requestedConveyorMode);
			
		SectionTask.ACTIVE, SectionTask.DISCHARGE:
			//once previous bundle catches up, the conveyor that bundle sits on must be linked to this section
			//a conveyor control module will handle linking
			
			IF conveyorsArr[i]^.IsOccupied THEN //follow this section's request
				conveyorsArr[i]^.setRequest(requestedConveyorMode);
				
			ELSE //catch up succeeding bundle (FOLLOW PREVIOUS SECTION)
				IF prevSection <> 0 THEN
					conveyorsArr[i]^.setRequest( prevSection^.pConveyorMode );
				END_IF
			END_IF
	END_CASE	
	
END_FOR
END_SET
END_PROPERTY

METHOD PROTECTED ABSTRACT process : BOOL
VAR_INPUT
	auto : BOOL;
END_VAR
VAR_OUTPUT
	error : BOOL;
END_VAR
(*
this method is implemented by each section according to their material packaging steps
*)
END_METHOD

METHOD PROTECTED ABSTRACT ps_AbortCondition : BOOL
VAR_INPUT
END_VAR
END_METHOD

METHOD PROTECTED ABSTRACT ps_Aborted : BOOL
VAR_INPUT
END_VAR
END_METHOD

METHOD PROTECTED ABSTRACT ps_Aborting : BOOL
VAR_INPUT
END_VAR
END_METHOD

METHOD PROTECTED ABSTRACT ps_Clearing : BOOL
VAR_INPUT
END_VAR
END_METHOD

METHOD PROTECTED ABSTRACT ps_Complete : BOOL
VAR_INPUT
END_VAR
END_METHOD

METHOD PROTECTED ABSTRACT ps_Completing : BOOL
VAR_INPUT
END_VAR
END_METHOD

METHOD PROTECTED FINAL ps_Execute : BOOL
VAR_INPUT
END_VAR
VAR_OUTPUT
	error : BOOL;
END_VAR
CASE pmlMode OF
	0: //invalid mode
	ePMLCustomUnitMode_Production:		ps_Execute := runSectionTasks(auto := TRUE);
	ePMLCustomUnitMode_Maintenance:		ps_Execute := maintenance();
	ePMLCustomUnitMode_Manual:			ps_Execute := manual();
	ePMLCustomUnitMode_SemiAuto:		ps_Execute := runSectionTasks(auto := FALSE);
END_CASE
END_METHOD

METHOD PROTECTED ABSTRACT ps_Held : BOOL
VAR_INPUT
END_VAR
END_METHOD

METHOD PROTECTED ABSTRACT ps_HoldCondition : BOOL
VAR_INPUT
END_VAR
END_METHOD

METHOD PROTECTED ABSTRACT ps_Holding : BOOL
VAR_INPUT
END_VAR
END_METHOD

METHOD PROTECTED FINAL ps_Idle : BOOL
VAR_INPUT
END_VAR
ps_Idle := run := run OR trigger.Q; (*start section input*)
END_METHOD

METHOD PROTECTED ABSTRACT ps_Resetting : BOOL
VAR_INPUT
END_VAR
END_METHOD

METHOD PROTECTED ABSTRACT ps_Starting : BOOL
VAR_INPUT
END_VAR
END_METHOD

METHOD PROTECTED ABSTRACT ps_StopCondition : BOOL
VAR_INPUT
END_VAR
END_METHOD

METHOD PROTECTED ABSTRACT ps_Stopped : BOOL
VAR_INPUT
END_VAR
END_METHOD

METHOD PROTECTED ABSTRACT ps_Stopping : BOOL
VAR_INPUT
END_VAR
END_METHOD

METHOD PROTECTED ABSTRACT ps_SuspendCondition : BOOL
VAR_INPUT
END_VAR
END_METHOD

METHOD PROTECTED ABSTRACT ps_Suspended : BOOL
VAR_INPUT
END_VAR
END_METHOD

METHOD PROTECTED ABSTRACT ps_Suspending : BOOL
VAR_INPUT
END_VAR
END_METHOD

METHOD PROTECTED ABSTRACT ps_Unholding : BOOL
VAR_INPUT
END_VAR
END_METHOD

METHOD PROTECTED ABSTRACT ps_Unsuspending : BOOL
VAR_INPUT
END_VAR
END_METHOD

METHOD PROTECTED runSectionTasks : BOOL
VAR_INPUT
	auto : BOOL;
END_VAR
VAR_OUTPUT
	error : BOOL;
END_VAR
CASE status OF
	SectionTask.IDLE:
		IF BundleIsValid(currentBundle) THEN			
			status := SectionTask.ALIGN;
			done := FALSE;
		END_IF
	
	SectionTask.ALIGN:		
		pConveyorMode := ConveyorMode.FORWARD;
		
		IF occupied THEN
			(*
			from here, there are 2 possible events:
				the expected bundle has arrived - proceed as normal
				a previously completed bundle backed up into this section - store the current position as 0 and go to STATUS -100
			*)
			pConveyorMode := ConveyorMode.STOP;
			
			IF nextSection <> 0 AND_THEN nextSection^.pConveyorMode = ConveyorMode.BACKWARD THEN
				status := -100;
				
			ELSIF NOT auto OR_ELSE trigger.Q THEN
				//zero the conveyors again
				status := SectionTask.ACTIVE;
				
			END_IF
		END_IF
		
	SectionTask.ACTIVE:
		activeBundle := currentBundle;
		
		IF NOT enable THEN
			iPair := 0;
			status := SectionTask.DISCHARGE;
			
		ELSIF currentBundle.bypass (*AND_THEN discharge()*) THEN //bundle failed in previous section, discharge this section's materials
			IF unload() THEN
				iPair := 0;
				status := SectionTask.DISCHARGE;
			END_IF
			
		ELSIF process(auto := auto, error => error) THEN //bundle recipe completed normally
			IF NOT auto OR_ELSE trigger.Q THEN
				iPair := 0;
				status := SectionTask.DISCHARGE;
			END_IF			
		END_IF
		
	SectionTask.DISCHARGE:
		activeBundle := currentBundle;
		pConveyorMode := ConveyorMode.FORWARD;
		
